LIN {X 0,Y 424.984,Z 508.898,A -85,B 0,C 180,E1 -17595.591,E2 -17595.591} C_VEL
LIN {X 0,Y 428.551,Z 453.272,A -85,B 0,C 180,E1 -17596.618,E2 -17596.618} C_VEL
LIN {X 0,Y 430.849,Z 412.705,A -85,B 0,C 180,E1 -17597.315,E2 -17597.315} C_VEL
LIN {X 0,Y 437.854,Z 381.493,A -85,B 0,C 180,E1 -17598.457,E2 -17598.457} C_VEL
LIN {X 0,Y 438.102,Z 374.288,A -85,B 0,C 180,E1 -17598.991,E2 -17598.991} C_VEL
LIN {X 0,Y 431.7,Z 356.101,A -85,B 0,C 180,E1 -17601.63,E2 -17601.63} C_VEL
LIN {X 0,Y 425.544,Z 340.551,A -85,B 0,C 180,E1 -17604.192,E2 -17604.192} C_VEL
LIN {X 0,Y 418.875,Z 325.42,A -85,B 0,C 180,E1 -17607.026,E2 -17607.026} C_VEL
LIN {X 0,Y 411.539,Z 310.81,A -85,B 0,C 180,E1 -17610.127,E2 -17610.127} C_VEL
LIN {X 0,Y 405.656,Z 300.356,A -85,B 0,C 180,E1 -17612.712,E2 -17612.712} C_VEL
LIN {X 0,Y 401.04,Z 292.309,A -85,B 0,C 180,E1 -17614.922,E2 -17614.922} C_VEL
LIN {X 0,Y 397.213,Z 286.474,A -85,B 0,C 180,E1 -17616.721,E2 -17616.721} C_VEL
LIN {X 0,Y 394.441,Z 281.986,A -85,B 0,C 180,E1 -17618.2,E2 -17618.2} C_VEL
LIN {X 0,Y 391.017,Z 276.874,A -85,B 0,C 180,E1 -17620.039,E2 -17620.039} C_VEL
LIN {X 0,Y 388.14,Z 272.719,A -85,B 0,C 180,E1 -17621.721,E2 -17621.721} C_VEL
LIN {X 0,Y 387.304,Z 271.349,A -85,B 0,C 180,E1 -17622.264,E2 -17622.264} C_VEL
LIN {X 0,Y 384.465,Z 267.744,A -85,B 0,C 180,E1 -17624.075,E2 -17624.075} C_VEL
LIN {X 0,Y 383.391,Z 265.721,A -85,B 0,C 180,E1 -17624.882,E2 -17624.882} C_VEL
LIN {X 0,Y 380.512,Z 262.705,A -85,B 0,C 180,E1 -17626.939,E2 -17626.939} C_VEL
LIN {X 0,Y 379.113,Z 259.666,A -85,B 0,C 180,E1 -17628.283,E2 -17628.283} C_VEL
LIN {X 0,Y 375.9,Z 257.035,A -85,B 0,C 180,E1 -17631.125,E2 -17631.125} C_VEL
LIN {X 0,Y 374.343,Z 253.325,A -85,B 0,C 180,E1 -17633.405,E2 -17633.405} C_VEL
LIN {X 0,Y 370.867,Z 250.89,A -85,B 0,C 180,E1 -17641.236,E2 -17641.236} C_VEL
LIN {X 0,Y 371.49,Z 251.549,A -85,B 0,C 180,E1 -17645.87,E2 -17645.87} C_VEL
LIN {X 0,Y 374.488,Z 253.671,A -85,B 0,C 180,E1 -17650.729,E2 -17650.729} C_VEL
LIN {X 0,Y 376.122,Z 261.606,A -85,B 0,C 180,E1 -17653.647,E2 -17653.647} C_VEL
LIN {X 0,Y 378.615,Z 269.925,A -85,B 0,C 180,E1 -17656.414,E2 -17656.414} C_VEL
LIN {X 0,Y 385.424,Z 282.96,A -85,B 0,C 180,E1 -17659.71,E2 -17659.71} C_VEL
LIN {X 0,Y 393.512,Z 298.865,A -85,B 0,C 180,E1 -17663.353,E2 -17663.353} C_VEL
LIN {X 0,Y 402.331,Z 316.84,A -85,B 0,C 180,E1 -17667.052,E2 -17667.052} C_VEL
LIN {X 0,Y 410.157,Z 332.928,A -85,B 0,C 180,E1 -17670.004,E2 -17670.004} C_VEL
LIN {X 0,Y 428.238,Z 360.802,A -85,B 0,C 180,E1 -17673.138,E2 -17673.138} C_VEL
LIN {X 0,Y 436.471,Z 374.047,A -85,B 0,C 180,E1 -17674.486,E2 -17674.486} C_VEL
LIN {X 0,Y 417.243,Z 631.491,A -85,B 0,C 180,E1 -17679.901,E2 -17679.901} C_VEL
LIN {X 0,Y 412.894,Z 693.948,A -85,B 0,C 180,E1 -17681.283,E2 -17681.283} C_VEL
LIN {X 0,Y 410.167,Z 718.357,A -85,B 0,C 180,E1 -17682.04,E2 -17682.04} C_VEL
LIN {X 0,Y 406.626,Z 743.879,A -85,B 0,C 180,E1 -17683.087,E2 -17683.087} C_VEL
LIN {X 0,Y 402.884,Z 766.939,A -85,B 0,C 180,E1 -17684.276,E2 -17684.276} C_VEL
LIN {X 0,Y 398.654,Z 789.481,A -85,B 0,C 180,E1 -17685.718,E2 -17685.718} C_VEL
LIN {X 0,Y 393.831,Z 812.889,A -85,B 0,C 180,E1 -17687.519,E2 -17687.519} C_VEL
LIN {X 0,Y 389.308,Z 833.205,A -85,B 0,C 180,E1 -17689.377,E2 -17689.377} C_VEL
LIN {X 0,Y 384.718,Z 852.523,A -85,B 0,C 180,E1 -17691.473,E2 -17691.473} C_VEL
LIN {X 0,Y 380.138,Z 871.424,A -85,B 0,C 180,E1 -17693.854,E2 -17693.854} C_VEL
LIN {X 0,Y 375.883,Z 888.627,A -85,B 0,C 180,E1 -17696.406,E2 -17696.406} C_VEL
LIN {X 0,Y 371.678,Z 905.948,A -85,B 0,C 180,E1 -17699.414,E2 -17699.414} C_VEL
LIN {X 0,Y 368.526,Z 919.642,A -85,B 0,C 180,E1 -17702.192,E2 -17702.192} C_VEL
LIN {X 0,Y 365.762,Z 932.567,A -85,B 0,C 180,E1 -17705.275,E2 -17705.275} C_VEL
LIN {X 0,Y 363.603,Z 944.291,A -85,B 0,C 180,E1 -17708.547,E2 -17708.547} C_VEL
LIN {X 0,Y 362.169,Z 953.987,A -85,B 0,C 180,E1 -17711.822,E2 -17711.822} C_VEL
LIN {X 0,Y 361.326,Z 962.067,A -85,B 0,C 180,E1 -17715.087,E2 -17715.087} C_VEL
LIN {X 0,Y 360.957,Z 968.703,A -85,B 0,C 180,E1 -17718.495,E2 -17718.495} C_VEL
LIN {X 0,Y 360.949,Z 973.188,A -85,B 0,C 180,E1 -17721.477,E2 -17721.477} C_VEL
LIN {X 0,Y 361.102,Z 976.867,A -85,B 0,C 180,E1 -17724.917,E2 -17724.917} C_VEL
LIN {X 0,Y 361.251,Z 978.684,A -85,B 0,C 180,E1 -17728.097,E2 -17728.097} C_VEL
LIN {X 0,Y 361.231,Z 979.16,A -85,B 0,C 180,E1 -17730.952,E2 -17730.952} C_VEL
LIN {X 0,Y 361.074,Z 978.468,A -85,B 0,C 180,E1 -17733.97,E2 -17733.97} C_VEL
LIN {X 0,Y 360.804,Z 976.089,A -85,B 0,C 180,E1 -17737.484,E2 -17737.484} C_VEL
LIN {X 0,Y 360.711,Z 972.725,A -85,B 0,C 180,E1 -17740.542,E2 -17740.542} C_VEL
LIN {X 0,Y 360.927,Z 967.69,A -85,B 0,C 180,E1 -17743.947,E2 -17743.947} C_VEL
LIN {X 0,Y 361.857,Z 960.075,A -85,B 0,C 180,E1 -17747.862,E2 -17747.862} C_VEL
LIN {X 0,Y 363.44,Z 951.875,A -85,B 0,C 180,E1 -17751.294,E2 -17751.294} C_VEL
LIN {X 0,Y 366.317,Z 940.57,A -85,B 0,C 180,E1 -17755.202,E2 -17755.202} C_VEL
LIN {X 0,Y 370.299,Z 927.832,A -85,B 0,C 180,E1 -17758.904,E2 -17758.904} C_VEL
LIN {X 0,Y 375.296,Z 913.565,A -85,B 0,C 180,E1 -17762.379,E2 -17762.379} C_VEL
LIN {X 0,Y 381.882,Z 896.522,A -85,B 0,C 180,E1 -17765.91,E2 -17765.91} C_VEL
LIN {X 0,Y 389.169,Z 878.862,A -85,B 0,C 180,E1 -17769.012,E2 -17769.012} C_VEL
LIN {X 0,Y 397.276,Z 859.703,A -85,B 0,C 180,E1 -17771.841,E2 -17771.841} C_VEL
LIN {X 0,Y 406.471,Z 838.288,A -85,B 0,C 180,E1 -17774.514,E2 -17774.514} C_VEL
LIN {X 0,Y 416.369,Z 815.377,A -85,B 0,C 180,E1 -17776.89,E2 -17776.89} C_VEL
LIN {X 0,Y 425.924,Z 793.069,A -85,B 0,C 180,E1 -17778.799,E2 -17778.799} C_VEL
LIN {X 0,Y 435.049,Z 771.007,A -85,B 0,C 180,E1 -17780.349,E2 -17780.349} C_VEL
LIN {X 0,Y 443.884,Z 748.687,A -85,B 0,C 180,E1 -17781.619,E2 -17781.619} C_VEL
LIN {X 0,Y 448.557,Z 736.3,A -85,B 0,C 180,E1 -17782.233,E2 -17782.233} C_VEL
LIN {X 0,Y 438.455,Z 757.223,A -85,B 0,C 180,E1 -17783.472,E2 -17783.472} C_VEL
LIN {X 0,Y 428.026,Z 777.505,A -85,B 0,C 180,E1 -17785.005,E2 -17785.005} C_VEL
LIN {X 0,Y 417.47,Z 797.566,A -85,B 0,C 180,E1 -17786.901,E2 -17786.901} C_VEL
LIN {X 0,Y 407.438,Z 816.792,A -85,B 0,C 180,E1 -17789.142,E2 -17789.142} C_VEL
LIN {X 0,Y 398.353,Z 834.637,A -85,B 0,C 180,E1 -17791.679,E2 -17791.679} C_VEL
LIN {X 0,Y 390.604,Z 850.206,A -85,B 0,C 180,E1 -17794.366,E2 -17794.366} C_VEL
LIN {X 0,Y 384.339,Z 862.875,A -85,B 0,C 180,E1 -17797.031,E2 -17797.031} C_VEL
LIN {X 0,Y 379.023,Z 873.475,A -85,B 0,C 180,E1 -17799.782,E2 -17799.782} C_VEL
LIN {X 0,Y 374.57,Z 882.04,A -85,B 0,C 180,E1 -17802.604,E2 -17802.604} C_VEL
LIN {X 0,Y 370.918,Z 888.625,A -85,B 0,C 180,E1 -17805.481,E2 -17805.481} C_VEL
LIN {X 0,Y 368.15,Z 893.065,A -85,B 0,C 180,E1 -17808.247,E2 -17808.247} C_VEL
LIN {X 0,Y 366.013,Z 895.825,A -85,B 0,C 180,E1 -17811.042,E2 -17811.042} C_VEL
LIN {X 0,Y 364.426,Z 896.884,A -85,B 0,C 180,E1 -17813.857,E2 -17813.857} C_VEL
LIN {X 0,Y 363.265,Z 896.126,A -85,B 0,C 180,E1 -17816.844,E2 -17816.844} C_VEL
LIN {X 0,Y 362.594,Z 893.619,A -85,B 0,C 180,E1 -17819.684,E2 -17819.684} C_VEL
LIN {X 0,Y 362.254,Z 889.408,A -85,B 0,C 180,E1 -17822.531,E2 -17822.531} C_VEL
LIN {X 0,Y 362.232,Z 883.769,A -85,B 0,C 180,E1 -17825.226,E2 -17825.226} C_VEL
LIN {X 0,Y 362.532,Z 875.956,A -85,B 0,C 180,E1 -17828.086,E2 -17828.086} C_VEL
LIN {X 0,Y 363.206,Z 866.063,A -85,B 0,C 180,E1 -17830.95,E2 -17830.95} C_VEL
LIN {X 0,Y 364.27,Z 854.546,A -85,B 0,C 180,E1 -17833.663,E2 -17833.663} C_VEL
LIN {X 0,Y 365.672,Z 841.577,A -85,B 0,C 180,E1 -17836.195,E2 -17836.195} C_VEL
LIN {X 0,Y 367.459,Z 826.606,A -85,B 0,C 180,E1 -17838.647,E2 -17838.647} C_VEL
LIN {X 0,Y 369.541,Z 810.047,A -85,B 0,C 180,E1 -17840.926,E2 -17840.926} C_VEL
LIN {X 0,Y 371.846,Z 791.943,A -85,B 0,C 180,E1 -17843.012,E2 -17843.012} C_VEL
LIN {X 0,Y 374.252,Z 772.49,A -85,B 0,C 180,E1 -17844.885,E2 -17844.885} C_VEL
LIN {X 0,Y 376.791,Z 751.357,A -85,B 0,C 180,E1 -17846.561,E2 -17846.561} C_VEL
LIN {X 0,Y 379.246,Z 729.129,A -85,B 0,C 180,E1 -17847.989,E2 -17847.989} C_VEL
LIN {X 0,Y 381.469,Z 706.375,A -85,B 0,C 180,E1 -17849.137,E2 -17849.137} C_VEL
LIN {X 0,Y 383.428,Z 682.672,A -85,B 0,C 180,E1 -17850.019,E2 -17850.019} C_VEL
LIN {X 0,Y 395.248,Z 511.536,A -85,B 0,C 180,E1 -17854.648,E2 -17854.648} C_VEL
LIN {X 0,Y 391.838,Z 447.433,A -85,B 0,C 180,E1 -17857.121,E2 -17857.121} C_VEL
LIN {X 0,Y 393.218,Z 446.968,A -85,B 0,C 180,E1 -17857.381,E2 -17857.381} C_VEL
LIN {X 0,Y 395.398,Z 443.797,A -85,B 0,C 180,E1 -17857.71,E2 -17857.71} C_VEL
LIN {X 0,Y 398.815,Z 435.862,A -85,B 0,C 180,E1 -17858.126,E2 -17858.126} C_VEL
LIN {X 0,Y 400.426,Z 433.355,A -85,B 0,C 180,E1 -17858.354,E2 -17858.354} C_VEL
LIN {X 0,Y 404.177,Z 431.028,A -85,B 0,C 180,E1 -17858.976,E2 -17858.976} C_VEL
LIN {X 0,Y 408.609,Z 426.161,A -85,B 0,C 180,E1 -17859.626,E2 -17859.626} C_VEL
LIN {X 0,Y 409.577,Z 425.061,A -85,B 0,C 180,E1 -17859.763,E2 -17859.763} C_VEL
LIN {X 0,Y 414.152,Z 421.888,A -85,B 0,C 180,E1 -17860.455,E2 -17860.455} C_VEL
LIN {X 0,Y 418.92,Z 417.332,A -85,B 0,C 180,E1 -17861.025,E2 -17861.025} C_VEL
LIN {X 0,Y 423.934,Z 414.013,A -85,B 0,C 180,E1 -17861.692,E2 -17861.692} C_VEL
LIN {X 0,Y 428.557,Z 410.023,A -85,B 0,C 180,E1 -17862.218,E2 -17862.218} C_VEL
LIN {X 0,Y 431.714,Z 408.162,A -85,B 0,C 180,E1 -17862.628,E2 -17862.628} C_VEL
LIN {X 0,Y 430.489,Z 414.914,A -85,B 0,C 180,E1 -17862.841,E2 -17862.841} C_VEL
LIN {X 0,Y 425.936,Z 494.183,A -85,B 0,C 180,E1 -17864.222,E2 -17864.222} C_VEL
LIN {X 0,Y 421.205,Z 553.034,A -85,B 0,C 180,E1 -17865.466,E2 -17865.466} C_VEL
LIN {X 0,Y 415.261,Z 612.433,A -85,B 0,C 180,E1 -17866.95,E2 -17866.95} C_VEL
LIN {X 0,Y 410.707,Z 656.621,A -85,B 0,C 180,E1 -17868.27,E2 -17868.27} C_VEL
LIN {X 0,Y 408.041,Z 685.292,A -85,B 0,C 180,E1 -17869.326,E2 -17869.326} C_VEL
LIN {X 0,Y 405.524,Z 705.596,A -85,B 0,C 180,E1 -17870.312,E2 -17870.312} C_VEL
LIN {X 0,Y 402.242,Z 726.337,A -85,B 0,C 180,E1 -17871.578,E2 -17871.578} C_VEL
LIN {X 0,Y 398.508,Z 746.053,A -85,B 0,C 180,E1 -17873.064,E2 -17873.064} C_VEL
LIN {X 0,Y 394.229,Z 765.506,A -85,B 0,C 180,E1 -17874.848,E2 -17874.848} C_VEL
LIN {X 0,Y 389.705,Z 783.802,A -85,B 0,C 180,E1 -17876.872,E2 -17876.872} C_VEL
LIN {X 0,Y 385.137,Z 800.764,A -85,B 0,C 180,E1 -17879.122,E2 -17879.122} C_VEL
LIN {X 0,Y 380.552,Z 816.747,A -85,B 0,C 180,E1 -17881.668,E2 -17881.668} C_VEL
LIN {X 0,Y 376.385,Z 830.752,A -85,B 0,C 180,E1 -17884.341,E2 -17884.341} C_VEL
LIN {X 0,Y 372.544,Z 843.468,A -85,B 0,C 180,E1 -17887.264,E2 -17887.264} C_VEL
LIN {X 0,Y 369.226,Z 854.588,A -85,B 0,C 180,E1 -17890.379,E2 -17890.379} C_VEL
LIN {X 0,Y 366.629,Z 863.669,A -85,B 0,C 180,E1 -17893.523,E2 -17893.523} C_VEL
LIN {X 0,Y 364.673,Z 871.061,A -85,B 0,C 180,E1 -17896.749,E2 -17896.749} C_VEL
LIN {X 0,Y 363.308,Z 876.769,A -85,B 0,C 180,E1 -17900.015,E2 -17900.015} C_VEL
LIN {X 0,Y 362.432,Z 881.033,A -85,B 0,C 180,E1 -17903.505,E2 -17903.505} C_VEL
LIN {X 0,Y 362.034,Z 883.325,A -85,B 0,C 180,E1 -17906.583,E2 -17906.583} C_VEL
LIN {X 0,Y 360.957,Z 883.954,A -85,B 0,C 180,E1 -17907.799,E2 -17907.799} C_VEL
LIN {X 0,Y 354.617,Z 885.109,A -85,B 0,C 180,E1 -17911.143,E2 -17911.143} C_VEL
LIN {X 0,Y 354.012,Z 884.908,A -85,B 0,C 180,E1 -17912.13,E2 -17912.13} C_VEL
LIN {X 0,Y 354.34,Z 883.134,A -85,B 0,C 180,E1 -17915.505,E2 -17915.505} C_VEL
LIN {X 0,Y 355.032,Z 879.694,A -85,B 0,C 180,E1 -17918.911,E2 -17918.911} C_VEL
LIN {X 0,Y 356.194,Z 874.854,A -85,B 0,C 180,E1 -17922.154,E2 -17922.154} C_VEL
LIN {X 0,Y 358.029,Z 868.036,A -85,B 0,C 180,E1 -17925.551,E2 -17925.551} C_VEL
LIN {X 0,Y 360.466,Z 859.76,A -85,B 0,C 180,E1 -17928.77,E2 -17928.77} C_VEL
LIN {X 0,Y 363.449,Z 850.138,A -85,B 0,C 180,E1 -17931.802,E2 -17931.802} C_VEL
LIN {X 0,Y 367.117,Z 838.547,A -85,B 0,C 180,E1 -17934.799,E2 -17934.799} C_VEL
LIN {X 0,Y 371.487,Z 824.659,A -85,B 0,C 180,E1 -17937.752,E2 -17937.752} C_VEL
LIN {X 0,Y 376.128,Z 809.477,A -85,B 0,C 180,E1 -17940.426,E2 -17940.426} C_VEL
LIN {X 0,Y 380.722,Z 793.669,A -85,B 0,C 180,E1 -17942.753,E2 -17942.753} C_VEL
LIN {X 0,Y 385.565,Z 775.624,A -85,B 0,C 180,E1 -17944.968,E2 -17944.968} C_VEL
LIN {X 0,Y 390.072,Z 757.084,A -85,B 0,C 180,E1 -17946.857,E2 -17946.857} C_VEL
LIN {X 0,Y 394.24,Z 737.467,A -85,B 0,C 180,E1 -17948.51,E2 -17948.51} C_VEL
LIN {X 0,Y 397.983,Z 716.674,A -85,B 0,C 180,E1 -17949.935,E2 -17949.935} C_VEL
LIN {X 0,Y 401.085,Z 695.03,A -85,B 0,C 180,E1 -17951.117,E2 -17951.117} C_VEL
LIN {X 0,Y 403.458,Z 672.77,A -85,B 0,C 180,E1 -17952.049,E2 -17952.049} C_VEL
LIN {X 0,Y 407.778,Z 629.715,A -85,B 0,C 180,E1 -17953.455,E2 -17953.455} C_VEL
LIN {X 0,Y 414.06,Z 571.27,A -85,B 0,C 180,E1 -17955.005,E2 -17955.005} C_VEL
LIN {X 0,Y 419.279,Z 512.395,A -85,B 0,C 180,E1 -17956.318,E2 -17956.318} C_VEL
LIN {X 0,Y 422.898,Z 458.138,A -85,B 0,C 180,E1 -17957.334,E2 -17957.334} C_VEL
LIN {X 0,Y 425.379,Z 415.515,A -85,B 0,C 180,E1 -17958.07,E2 -17958.07} C_VEL
LIN {X 0,Y 432.668,Z 383.274,A -85,B 0,C 180,E1 -17959.238,E2 -17959.238} C_VEL
LIN {X 0,Y 432.805,Z 378.392,A -85,B 0,C 180,E1 -17959.607,E2 -17959.607} C_VEL
LIN {X 0,Y 426.533,Z 360.369,A -85,B 0,C 180,E1 -17962.277,E2 -17962.277} C_VEL
LIN {X 0,Y 420.306,Z 344.672,A -85,B 0,C 180,E1 -17964.921,E2 -17964.921} C_VEL
LIN {X 0,Y 413.62,Z 329.35,A -85,B 0,C 180,E1 -17967.871,E2 -17967.871} C_VEL
LIN {X 0,Y 407.095,Z 316.323,A -85,B 0,C 180,E1 -17970.74,E2 -17970.74} C_VEL
LIN {X 0,Y 401.641,Z 306.431,A -85,B 0,C 180,E1 -17973.217,E2 -17973.217} C_VEL
LIN {X 0,Y 397.019,Z 298.327,A -85,B 0,C 180,E1 -17975.525,E2 -17975.525} C_VEL
LIN {X 0,Y 393.875,Z 293.356,A -85,B 0,C 180,E1 -17977.066,E2 -17977.066} C_VEL
LIN {X 0,Y 391.222,Z 288.934,A -85,B 0,C 180,E1 -17978.563,E2 -17978.563} C_VEL
LIN {X 0,Y 387.999,Z 284.027,A -85,B 0,C 180,E1 -17980.348,E2 -17980.348} C_VEL
LIN {X 0,Y 385.133,Z 279.626,A -85,B 0,C 180,E1 -17982.121,E2 -17982.121} C_VEL
LIN {X 0,Y 381.484,Z 274.487,A -85,B 0,C 180,E1 -17984.571,E2 -17984.571} C_VEL
LIN {X 0,Y 380.825,Z 273.211,A -85,B 0,C 180,E1 -17985.09,E2 -17985.09} C_VEL
LIN {X 0,Y 377.944,Z 270.024,A -85,B 0,C 180,E1 -17987.238,E2 -17987.238} C_VEL
LIN {X 0,Y 376.766,Z 267.259,A -85,B 0,C 180,E1 -17988.519,E2 -17988.519} C_VEL
LIN {X 0,Y 373.477,Z 264.326,A -85,B 0,C 180,E1 -17991.532,E2 -17991.532} C_VEL
LIN {X 0,Y 372.123,Z 260.992,A -85,B 0,C 180,E1 -17993.675,E2 -17993.675} C_VEL
LIN {X 0,Y 369.027,Z 258.675,A -85,B 0,C 180,E1 -18001.242,E2 -18001.242} C_VEL
LIN {X 0,Y 369.744,Z 259.37,A -85,B 0,C 180,E1 -18005.898,E2 -18005.898} C_VEL
LIN {X 0,Y 372.489,Z 261.356,A -85,B 0,C 180,E1 -18010.439,E2 -18010.439} C_VEL
LIN {X 0,Y 373.965,Z 268.68,A -85,B 0,C 180,E1 -18013.176,E2 -18013.176} C_VEL
LIN {X 0,Y 376.51,Z 277.821,A -85,B 0,C 180,E1 -18016.191,E2 -18016.191} C_VEL
LIN {X 0,Y 381.85,Z 292.334,A -85,B 0,C 180,E1 -18020.381,E2 -18020.381} C_VEL
LIN {X 0,Y 390.043,Z 308.671,A -85,B 0,C 180,E1 -18024.054,E2 -18024.054} C_VEL
LIN {X 0,Y 399.158,Z 327.437,A -85,B 0,C 180,E1 -18027.839,E2 -18027.839} C_VEL
LIN {X 0,Y 402.379,Z 333.924,A -85,B 0,C 180,E1 -18029.01,E2 -18029.01} C_VEL
LIN {X 0,Y 422.571,Z 365.09,A -85,B 0,C 180,E1 -18032.601,E2 -18032.601} C_VEL
LIN {X 0,Y 430.139,Z 377.336,A -85,B 0,C 180,E1 -18033.862,E2 -18033.862} C_VEL
LIN {X 0,Y 410.702,Z 628.411,A -85,B 0,C 180,E1 -18039.24,E2 -18039.24} C_VEL
LIN {X 0,Y 405.985,Z 693.922,A -85,B 0,C 180,E1 -18040.718,E2 -18040.718} C_VEL
LIN {X 0,Y 403.21,Z 718.115,A -85,B 0,C 180,E1 -18041.482,E2 -18041.482} C_VEL
LIN {X 0,Y 399.697,Z 742.919,A -85,B 0,C 180,E1 -18042.511,E2 -18042.511} C_VEL
LIN {X 0,Y 395.798,Z 766.429,A -85,B 0,C 180,E1 -18043.738,E2 -18043.738} C_VEL
LIN {X 0,Y 391.526,Z 788.691,A -85,B 0,C 180,E1 -18045.182,E2 -18045.182} C_VEL
LIN {X 0,Y 386.728,Z 811.509,A -85,B 0,C 180,E1 -18046.955,E2 -18046.955} C_VEL
LIN {X 0,Y 382.094,Z 831.899,A -85,B 0,C 180,E1 -18048.842,E2 -18048.842} C_VEL
LIN {X 0,Y 377.316,Z 851.634,A -85,B 0,C 180,E1 -18051.002,E2 -18051.002} C_VEL
LIN {X 0,Y 372.803,Z 869.858,A -85,B 0,C 180,E1 -18053.317,E2 -18053.317} C_VEL
LIN {X 0,Y 368.526,Z 886.743,A -85,B 0,C 180,E1 -18055.846,E2 -18055.846} C_VEL
LIN {X 0,Y 364.361,Z 903.466,A -85,B 0,C 180,E1 -18058.758,E2 -18058.758} C_VEL
LIN {X 0,Y 361.088,Z 917.18,A -85,B 0,C 180,E1 -18061.557,E2 -18061.557} C_VEL
LIN {X 0,Y 358.024,Z 931.1,A -85,B 0,C 180,E1 -18064.881,E2 -18064.881} C_VEL
LIN {X 0,Y 355.871,Z 942.358,A -85,B 0,C 180,E1 -18068.057,E2 -18068.057} C_VEL
LIN {X 0,Y 354.277,Z 952.735,A -85,B 0,C 180,E1 -18071.573,E2 -18071.573} C_VEL
LIN {X 0,Y 353.4,Z 960.861,A -85,B 0,C 180,E1 -18074.912,E2 -18074.912} C_VEL
LIN {X 0,Y 353.012,Z 967.793,A -85,B 0,C 180,E1 -18078.531,E2 -18078.531} C_VEL
LIN {X 0,Y 353.017,Z 972.197,A -85,B 0,C 180,E1 -18081.53,E2 -18081.53} C_VEL
LIN {X 0,Y 353.177,Z 975.815,A -85,B 0,C 180,E1 -18084.965,E2 -18084.965} C_VEL
LIN {X 0,Y 353.328,Z 977.637,A -85,B 0,C 180,E1 -18088.216,E2 -18088.216} C_VEL
LIN {X 0,Y 353.299,Z 978.106,A -85,B 0,C 180,E1 -18091.135,E2 -18091.135} C_VEL
LIN {X 0,Y 353.106,Z 977.399,A -85,B 0,C 180,E1 -18094.222,E2 -18094.222} C_VEL
LIN {X 0,Y 352.83,Z 975.02,A -85,B 0,C 180,E1 -18097.818,E2 -18097.818} C_VEL
LIN {X 0,Y 352.727,Z 971.431,A -85,B 0,C 180,E1 -18101.114,E2 -18101.114} C_VEL
LIN {X 0,Y 353.03,Z 966.335,A -85,B 0,C 180,E1 -18104.601,E2 -18104.601} C_VEL
LIN {X 0,Y 354.059,Z 959.013,A -85,B 0,C 180,E1 -18108.439,E2 -18108.439} C_VEL
LIN {X 0,Y 355.906,Z 950.42,A -85,B 0,C 180,E1 -18112.115,E2 -18112.115} C_VEL
LIN {X 0,Y 359.099,Z 939.101,A -85,B 0,C 180,E1 -18116.1,E2 -18116.1} C_VEL
LIN {X 0,Y 363.454,Z 926.402,A -85,B 0,C 180,E1 -18119.864,E2 -18119.864} C_VEL
LIN {X 0,Y 368.927,Z 912.1,A -85,B 0,C 180,E1 -18123.408,E2 -18123.408} C_VEL
LIN {X 0,Y 375.947,Z 895.333,A -85,B 0,C 180,E1 -18126.948,E2 -18126.948} C_VEL
LIN {X 0,Y 383.727,Z 877.917,A -85,B 0,C 180,E1 -18130.062,E2 -18130.062} C_VEL
LIN {X 0,Y 392.756,Z 858.185,A -85,B 0,C 180,E1 -18133.023,E2 -18133.023} C_VEL
LIN {X 0,Y 402.833,Z 836.606,A -85,B 0,C 180,E1 -18135.734,E2 -18135.734} C_VEL
LIN {X 0,Y 413.334,Z 814.204,A -85,B 0,C 180,E1 -18138.062,E2 -18138.062} C_VEL
LIN {X 0,Y 423.737,Z 791.887,A -85,B 0,C 180,E1 -18139.971,E2 -18139.971} C_VEL
LIN {X 0,Y 433.523,Z 770.179,A -85,B 0,C 180,E1 -18141.484,E2 -18141.484} C_VEL
LIN {X 0,Y 439.331,Z 756.867,A -85,B 0,C 180,E1 -18142.29,E2 -18142.29} C_VEL
LIN {X 0,Y 428.322,Z 776.559,A -85,B 0,C 180,E1 -18143.716,E2 -18143.716} C_VEL
LIN {X 0,Y 416.856,Z 796.27,A -85,B 0,C 180,E1 -18145.522,E2 -18145.522} C_VEL
LIN {X 0,Y 405.872,Z 815.235,A -85,B 0,C 180,E1 -18147.684,E2 -18147.684} C_VEL
LIN {X 0,Y 395.858,Z 832.952,A -85,B 0,C 180,E1 -18150.159,E2 -18150.159} C_VEL
LIN {X 0,Y 387.233,Z 848.533,A -85,B 0,C 180,E1 -18152.804,E2 -18152.804} C_VEL
LIN {X 0,Y 379.645,Z 862.38,A -85,B 0,C 180,E1 -18155.683,E2 -18155.683} C_VEL
LIN {X 0,Y 373.638,Z 873.294,A -85,B 0,C 180,E1 -18158.492,E2 -18158.492} C_VEL
LIN {X 0,Y 368.676,Z 882.065,A -85,B 0,C 180,E1 -18161.335,E2 -18161.335} C_VEL
LIN {X 0,Y 364.771,Z 888.63,A -85,B 0,C 180,E1 -18164.091,E2 -18164.091} C_VEL
LIN {X 0,Y 361.266,Z 893.892,A -85,B 0,C 180,E1 -18167.208,E2 -18167.208} C_VEL
LIN {X 0,Y 358.703,Z 896.947,A -85,B 0,C 180,E1 -18170.21,E2 -18170.21} C_VEL
LIN {X 0,Y 356.898,Z 898.104,A -85,B 0,C 180,E1 -18173.081,E2 -18173.081} C_VEL
LIN {X 0,Y 355.611,Z 897.569,A -85,B 0,C 180,E1 -18175.969,E2 -18175.969} C_VEL
LIN {X 0,Y 354.79,Z 895.361,A -85,B 0,C 180,E1 -18178.87,E2 -18178.87} C_VEL
LIN {X 0,Y 354.351,Z 891.466,A -85,B 0,C 180,E1 -18181.779,E2 -18181.779} C_VEL
LIN {X 0,Y 354.245,Z 885.77,A -85,B 0,C 180,E1 -18184.695,E2 -18184.695} C_VEL
LIN {X 0,Y 354.468,Z 878.694,A -85,B 0,C 180,E1 -18187.456,E2 -18187.456} C_VEL
LIN {X 0,Y 355.018,Z 869.756,A -85,B 0,C 180,E1 -18190.221,E2 -18190.221} C_VEL
LIN {X 0,Y 355.971,Z 858.79,A -85,B 0,C 180,E1 -18192.986,E2 -18192.986} C_VEL
LIN {X 0,Y 357.29,Z 846.403,A -85,B 0,C 180,E1 -18195.585,E2 -18195.585} C_VEL
LIN {X 0,Y 358.979,Z 832.235,A -85,B 0,C 180,E1 -18198.081,E2 -18198.081} C_VEL
LIN {X 0,Y 360.984,Z 816.384,A -85,B 0,C 180,E1 -18200.427,E2 -18200.427} C_VEL
LIN {X 0,Y 363.327,Z 798.388,A -85,B 0,C 180,E1 -18202.662,E2 -18202.662} C_VEL
LIN {X 0,Y 365.876,Z 778.547,A -85,B 0,C 180,E1 -18204.717,E2 -18204.717} C_VEL
LIN {X 0,Y 368.373,Z 758.536,A -85,B 0,C 180,E1 -18206.433,E2 -18206.433} C_VEL
LIN {X 0,Y 370.948,Z 736.616,A -85,B 0,C 180,E1 -18207.971,E2 -18207.971} C_VEL
LIN {X 0,Y 373.29,Z 714.104,A -85,B 0,C 180,E1 -18209.221,E2 -18209.221} C_VEL
LIN {X 0,Y 375.438,Z 690.485,A -85,B 0,C 180,E1 -18210.222,E2 -18210.222} C_VEL
LIN {X 0,Y 378.003,Z 654.561,A -85,B 0,C 180,E1 -18211.312,E2 -18211.312} C_VEL
LIN {X 0,Y 388.249,Z 512.214,A -85,B 0,C 180,E1 -18215.216,E2 -18215.216} C_VEL
LIN {X 0,Y 386.223,Z 472.757,A -85,B 0,C 180,E1 -18216.776,E2 -18216.776} C_VEL
LIN {X 0,Y 387.587,Z 472.354,A -85,B 0,C 180,E1 -18217.041,E2 -18217.041} C_VEL
LIN {X 0,Y 389.842,Z 469.038,A -85,B 0,C 180,E1 -18217.39,E2 -18217.39} C_VEL
LIN {X 0,Y 392.918,Z 461.347,A -85,B 0,C 180,E1 -18217.759,E2 -18217.759} C_VEL
LIN {X 0,Y 395.267,Z 453.532,A -85,B 0,C 180,E1 -18217.977,E2 -18217.977} C_VEL
LIN {X 0,Y 398.142,Z 449.735,A -85,B 0,C 180,E1 -18218.409,E2 -18218.409} C_VEL
LIN {X 0,Y 401.43,Z 442.671,A -85,B 0,C 180,E1 -18218.811,E2 -18218.811} C_VEL
LIN {X 0,Y 402.505,Z 440.316,A -85,B 0,C 180,E1 -18218.939,E2 -18218.939} C_VEL
LIN {X 0,Y 407.194,Z 436.824,A -85,B 0,C 180,E1 -18219.676,E2 -18219.676} C_VEL
LIN {X 0,Y 411.77,Z 431.891,A -85,B 0,C 180,E1 -18220.326,E2 -18220.326} C_VEL
LIN {X 0,Y 417.125,Z 427.794,A -85,B 0,C 180,E1 -18221.103,E2 -18221.103} C_VEL
LIN {X 0,Y 421.231,Z 423.838,A -85,B 0,C 180,E1 -18221.655,E2 -18221.655} C_VEL
LIN {X 0,Y 424.807,Z 421.477,A -85,B 0,C 180,E1 -18222.151,E2 -18222.151} C_VEL
LIN {X 0,Y 420.272,Z 497.691,A -85,B 0,C 180,E1 -18223.49,E2 -18223.49} C_VEL
LIN {X 0,Y 415.453,Z 555.616,A -85,B 0,C 180,E1 -18224.729,E2 -18224.729} C_VEL
LIN {X 0,Y 409.469,Z 613.57,A -85,B 0,C 180,E1 -18226.194,E2 -18226.194} C_VEL
LIN {X 0,Y 404.775,Z 657.664,A -85,B 0,C 180,E1 -18227.528,E2 -18227.528} C_VEL
LIN {X 0,Y 401.93,Z 687.022,A -85,B 0,C 180,E1 -18228.627,E2 -18228.627} C_VEL
LIN {X 0,Y 399.248,Z 707.767,A -85,B 0,C 180,E1 -18229.654,E2 -18229.654} C_VEL
LIN {X 0,Y 395.858,Z 728.321,A -85,B 0,C 180,E1 -18230.934,E2 -18230.934} C_VEL
LIN {X 0,Y 392.003,Z 747.896,A -85,B 0,C 180,E1 -18232.438,E2 -18232.438} C_VEL
LIN {X 0,Y 387.583,Z 767.232,A -85,B 0,C 180,E1 -18234.244,E2 -18234.244} C_VEL
LIN {X 0,Y 382.853,Z 785.607,A -85,B 0,C 180,E1 -18236.318,E2 -18236.318} C_VEL
LIN {X 0,Y 378.121,Z 802.479,A -85,B 0,C 180,E1 -18238.604,E2 -18238.604} C_VEL
LIN {X 0,Y 373.387,Z 818.314,A -85,B 0,C 180,E1 -18241.182,E2 -18241.182} C_VEL
LIN {X 0,Y 368.975,Z 832.505,A -85,B 0,C 180,E1 -18243.959,E2 -18243.959} C_VEL
LIN {X 0,Y 364.997,Z 845.109,A -85,B 0,C 180,E1 -18246.937,E2 -18246.937} C_VEL
LIN {X 0,Y 361.557,Z 856.127,A -85,B 0,C 180,E1 -18250.113,E2 -18250.113} C_VEL
LIN {X 0,Y 358.734,Z 865.576,A -85,B 0,C 180,E1 -18253.501,E2 -18253.501} C_VEL
LIN {X 0,Y 356.696,Z 872.928,A -85,B 0,C 180,E1 -18256.876,E2 -18256.876} C_VEL
LIN {X 0,Y 355.302,Z 878.489,A -85,B 0,C 180,E1 -18260.279,E2 -18260.279} C_VEL
LIN {X 0,Y 354.473,Z 882.337,A -85,B 0,C 180,E1 -18263.684,E2 -18263.684} C_VEL
LIN {X 0,Y 354.056,Z 884.554,A -85,B 0,C 180,E1 -18267.086,E2 -18267.086} C_VEL
LIN {X 0,Y 353.956,Z 885.197,A -85,B 0,C 180,E1 -18270.324,E2 -18270.324} C_VEL
LIN {X 0,Y 354.012,Z 884.908,A -85,B 0,C 180,E1 -18272.13,E2 -18272.13} C_VEL
LIN {X 0,Y 353.105,Z 884.552,A -85,B 0,C 180,E1 -18273.378,E2 -18273.378} C_VEL
LIN {X 0,Y 347.381,Z 883.219,A -85,B 0,C 180,E1 -18276.728,E2 -18276.728} C_VEL
LIN {X 0,Y 346.846,Z 882.204,A -85,B 0,C 180,E1 -18277.815,E2 -18277.815} C_VEL
LIN {X 0,Y 347.975,Z 877.54,A -85,B 0,C 180,E1 -18281.436,E2 -18281.436} C_VEL
LIN {X 0,Y 349.824,Z 870.903,A -85,B 0,C 180,E1 -18285.076,E2 -18285.076} C_VEL
LIN {X 0,Y 352.418,Z 862.388,A -85,B 0,C 180,E1 -18288.623,E2 -18288.623} C_VEL
LIN {X 0,Y 355.68,Z 852.278,A -85,B 0,C 180,E1 -18291.956,E2 -18291.956} C_VEL
LIN {X 0,Y 359.439,Z 840.872,A -85,B 0,C 180,E1 -18295.014,E2 -18295.014} C_VEL
LIN {X 0,Y 363.671,Z 828.008,A -85,B 0,C 180,E1 -18297.866,E2 -18297.866} C_VEL
LIN {X 0,Y 367.962,Z 814.594,A -85,B 0,C 180,E1 -18300.36,E2 -18300.36} C_VEL
LIN {X 0,Y 372.603,Z 799.462,A -85,B 0,C 180,E1 -18302.733,E2 -18302.733} C_VEL
LIN {X 0,Y 377.344,Z 782.911,A -85,B 0,C 180,E1 -18304.915,E2 -18304.915} C_VEL
LIN {X 0,Y 381.724,Z 766.258,A -85,B 0,C 180,E1 -18306.765,E2 -18306.765} C_VEL
LIN {X 0,Y 385.962,Z 748.26,A -85,B 0,C 180,E1 -18308.444,E2 -18308.444} C_VEL
LIN {X 0,Y 389.967,Z 728.551,A -85,B 0,C 180,E1 -18309.963,E2 -18309.963} C_VEL
LIN {X 0,Y 393.455,Z 707.895,A -85,B 0,C 180,E1 -18311.25,E2 -18311.25} C_VEL
LIN {X 0,Y 396.308,Z 686.094,A -85,B 0,C 180,E1 -18312.318,E2 -18312.318} C_VEL
LIN {X 0,Y 399.857,Z 650.548,A -85,B 0,C 180,E1 -18313.613,E2 -18313.613} C_VEL
LIN {X 0,Y 405.349,Z 601.675,A -85,B 0,C 180,E1 -18315.044,E2 -18315.044} C_VEL
LIN {X 0,Y 410.919,Z 547.326,A -85,B 0,C 180,E1 -18316.384,E2 -18316.384} C_VEL
LIN {X 0,Y 415.551,Z 490.609,A -85,B 0,C 180,E1 -18317.569,E2 -18317.569} C_VEL
LIN {X 0,Y 419.979,Z 418.206,A -85,B 0,C 180,E1 -18318.845,E2 -18318.845} C_VEL
LIN {X 0,Y 427.547,Z 384.988,A -85,B 0,C 180,E1 -18320.04,E2 -18320.04} C_VEL
LIN {X 0,Y 427.552,Z 382.519,A -85,B 0,C 180,E1 -18320.236,E2 -18320.236} C_VEL
LIN {X 0,Y 421.414,Z 364.665,A -85,B 0,C 180,E1 -18322.939,E2 -18322.939} C_VEL
LIN {X 0,Y 415.15,Z 348.657,A -85,B 0,C 180,E1 -18325.702,E2 -18325.702} C_VEL
LIN {X 0,Y 408.377,Z 333.351,A -85,B 0,C 180,E1 -18328.73,E2 -18328.73} C_VEL
LIN {X 0,Y 402.415,Z 321.186,A -85,B 0,C 180,E1 -18331.506,E2 -18331.506} C_VEL
LIN {X 0,Y 396.611,Z 310.397,A -85,B 0,C 180,E1 -18334.302,E2 -18334.302} C_VEL
LIN {X 0,Y 391.135,Z 301.045,A -85,B 0,C 180,E1 -18337.134,E2 -18337.134} C_VEL
LIN {X 0,Y 388.021,Z 295.874,A -85,B 0,C 180,E1 -18338.932,E2 -18338.932} C_VEL
LIN {X 0,Y 384.994,Z 291.173,A -85,B 0,C 180,E1 -18340.662,E2 -18340.662} C_VEL
LIN {X 0,Y 382.188,Z 286.545,A -85,B 0,C 180,E1 -18342.53,E2 -18342.53} C_VEL
LIN {X 0,Y 378.955,Z 282.176,A -85,B 0,C 180,E1 -18344.701,E2 -18344.701} C_VEL
LIN {X 0,Y 378.03,Z 280.526,A -85,B 0,C 180,E1 -18345.447,E2 -18345.447} C_VEL
LIN {X 0,Y 375.234,Z 277.05,A -85,B 0,C 180,E1 -18347.691,E2 -18347.691} C_VEL
LIN {X 0,Y 374.296,Z 274.809,A -85,B 0,C 180,E1 -18348.755,E2 -18348.755} C_VEL
LIN {X 0,Y 371.321,Z 271.937,A -85,B 0,C 180,E1 -18351.717,E2 -18351.717} C_VEL
LIN {X 0,Y 370.039,Z 268.706,A -85,B 0,C 180,E1 -18353.795,E2 -18353.795} C_VEL
LIN {X 0,Y 367.154,Z 266.442,A -85,B 0,C 180,E1 -18361.404,E2 -18361.404} C_VEL
LIN {X 0,Y 368.011,Z 267.237,A -85,B 0,C 180,E1 -18366.083,E2 -18366.083} C_VEL
LIN {X 0,Y 370.532,Z 269.088,A -85,B 0,C 180,E1 -18370.181,E2 -18370.181} C_VEL
LIN {X 0,Y 371.851,Z 275.876,A -85,B 0,C 180,E1 -18372.738,E2 -18372.738} C_VEL
LIN {X 0,Y 374.308,Z 285.032,A -85,B 0,C 180,E1 -18375.772,E2 -18375.772} C_VEL
LIN {X 0,Y 379.498,Z 300.184,A -85,B 0,C 180,E1 -18380.151,E2 -18380.151} C_VEL
LIN {X 0,Y 387.563,Z 319.875,A -85,B 0,C 180,E1 -18384.868,E2 -18384.868} C_VEL
LIN {X 0,Y 394.603,Z 335.094,A -85,B 0,C 180,E1 -18387.996,E2 -18387.996} C_VEL
LIN {X 0,Y 411.937,Z 361.642,A -85,B 0,C 180,E1 -18391.193,E2 -18391.193} C_VEL
LIN {X 0,Y 423.773,Z 380.727,A -85,B 0,C 180,E1 -18393.234,E2 -18393.234} C_VEL
LIN {X 0,Y 403.08,Z 640.594,A -85,B 0,C 180,E1 -18398.906,E2 -18398.906} C_VEL
LIN {X 0,Y 398.994,Z 694.506,A -85,B 0,C 180,E1 -18400.166,E2 -18400.166} C_VEL
LIN {X 0,Y 396.142,Z 718.636,A -85,B 0,C 180,E1 -18400.946,E2 -18400.946} C_VEL
LIN {X 0,Y 392.53,Z 743.375,A -85,B 0,C 180,E1 -18401.998,E2 -18401.998} C_VEL
LIN {X 0,Y 388.52,Z 766.895,A -85,B 0,C 180,E1 -18403.254,E2 -18403.254} C_VEL
LIN {X 0,Y 383.956,Z 790.092,A -85,B 0,C 180,E1 -18404.795,E2 -18404.795} C_VEL
LIN {X 0,Y 379.079,Z 812.597,A -85,B 0,C 180,E1 -18406.598,E2 -18406.598} C_VEL
LIN {X 0,Y 374.178,Z 833.62,A -85,B 0,C 180,E1 -18408.595,E2 -18408.595} C_VEL
LIN {X 0,Y 369.316,Z 853.128,A -85,B 0,C 180,E1 -18410.81,E2 -18410.81} C_VEL
LIN {X 0,Y 364.284,Z 872.858,A -85,B 0,C 180,E1 -18413.443,E2 -18413.443} C_VEL
LIN {X 0,Y 359.737,Z 890.512,A -85,B 0,C 180,E1 -18416.21,E2 -18416.21} C_VEL
LIN {X 0,Y 355.626,Z 906.727,A -85,B 0,C 180,E1 -18419.222,E2 -18419.222} C_VEL
LIN {X 0,Y 352.112,Z 921.437,A -85,B 0,C 180,E1 -18422.428,E2 -18422.428} C_VEL
LIN {X 0,Y 349.518,Z 933.352,A -85,B 0,C 180,E1 -18425.493,E2 -18425.493} C_VEL
LIN {X 0,Y 347.327,Z 945.157,A -85,B 0,C 180,E1 -18429.086,E2 -18429.086} C_VEL
LIN {X 0,Y 346.043,Z 954.062,A -85,B 0,C 180,E1 -18432.338,E2 -18432.338} C_VEL
LIN {X 0,Y 345.258,Z 962.402,A -85,B 0,C 180,E1 -18436.092,E2 -18436.092} C_VEL
LIN {X 0,Y 345.051,Z 967.893,A -85,B 0,C 180,E1 -18439.222,E2 -18439.222} C_VEL
LIN {X 0,Y 345.124,Z 972.521,A -85,B 0,C 180,E1 -18442.676,E2 -18442.676} C_VEL
LIN {X 0,Y 345.329,Z 975.386,A -85,B 0,C 180,E1 -18446.015,E2 -18446.015} C_VEL
LIN {X 0,Y 345.409,Z 976.769,A -85,B 0,C 180,E1 -18449.005,E2 -18449.005} C_VEL
LIN {X 0,Y 345.305,Z 977.005,A -85,B 0,C 180,E1 -18452.157,E2 -18452.157} C_VEL
LIN {X 0,Y 345.046,Z 975.752,A -85,B 0,C 180,E1 -18455.654,E2 -18455.654} C_VEL
LIN {X 0,Y 344.799,Z 973.147,A -85,B 0,C 180,E1 -18459.009,E2 -18459.009} C_VEL
LIN {X 0,Y 344.817,Z 969.073,A -85,B 0,C 180,E1 -18462.561,E2 -18462.561} C_VEL
LIN {X 0,Y 345.466,Z 962.594,A -85,B 0,C 180,E1 -18466.651,E2 -18466.651} C_VEL
LIN {X 0,Y 346.892,Z 955.072,A -85,B 0,C 180,E1 -18470.412,E2 -18470.412} C_VEL
LIN {X 0,Y 349.593,Z 944.98,A -85,B 0,C 180,E1 -18474.502,E2 -18474.502} C_VEL
LIN {X 0,Y 353.495,Z 933.505,A -85,B 0,C 180,E1 -18478.394,E2 -18478.394} C_VEL
LIN {X 0,Y 358.699,Z 920.105,A -85,B 0,C 180,E1 -18482.169,E2 -18482.169} C_VEL
LIN {X 0,Y 365.389,Z 904.751,A -85,B 0,C 180,E1 -18485.847,E2 -18485.847} C_VEL
LIN {X 0,Y 373.195,Z 888.055,A -85,B 0,C 180,E1 -18489.221,E2 -18489.221} C_VEL
LIN {X 0,Y 381.941,Z 870.073,A -85,B 0,C 180,E1 -18492.284,E2 -18492.284} C_VEL
LIN {X 0,Y 392.294,Z 849.528,A -85,B 0,C 180,E1 -18495.223,E2 -18495.223} C_VEL
LIN {X 0,Y 402.876,Z 828.807,A -85,B 0,C 180,E1 -18497.698,E2 -18497.698} C_VEL
LIN {X 0,Y 414.345,Z 806.273,A -85,B 0,C 180,E1 -18499.905,E2 -18499.905} C_VEL
LIN {X 0,Y 425.952,Z 783.125,A -85,B 0,C 180,E1 -18501.741,E2 -18501.741} C_VEL
LIN {X 0,Y 430.183,Z 774.498,A -85,B 0,C 180,E1 -18502.337,E2 -18502.337} C_VEL
LIN {X 0,Y 417.846,Z 793.984,A -85,B 0,C 180,E1 -18504.022,E2 -18504.022} C_VEL
LIN {X 0,Y 406.069,Z 812.314,A -85,B 0,C 180,E1 -18506.016,E2 -18506.016} C_VEL
LIN {X 0,Y 394.907,Z 829.925,A -85,B 0,C 180,E1 -18508.391,E2 -18508.391} C_VEL
LIN {X 0,Y 384.787,Z 846.339,A -85,B 0,C 180,E1 -18511.097,E2 -18511.097} C_VEL
LIN {X 0,Y 376.157,Z 860.63,A -85,B 0,C 180,E1 -18513.985,E2 -18513.985} C_VEL
LIN {X 0,Y 369.175,Z 872.195,A -85,B 0,C 180,E1 -18516.876,E2 -18516.876} C_VEL
LIN {X 0,Y 363.564,Z 881.294,A -85,B 0,C 180,E1 -18519.725,E2 -18519.725} C_VEL
LIN {X 0,Y 358.867,Z 888.538,A -85,B 0,C 180,E1 -18522.655,E2 -18522.655} C_VEL
LIN {X 0,Y 355.002,Z 893.969,A -85,B 0,C 180,E1 -18525.674,E2 -18525.674} C_VEL
LIN {X 0,Y 352.008,Z 897.518,A -85,B 0,C 180,E1 -18528.697,E2 -18528.697} C_VEL
LIN {X 0,Y 349.838,Z 899.205,A -85,B 0,C 180,E1 -18531.618,E2 -18531.618} C_VEL
LIN {X 0,Y 348.25,Z 899.262,A -85,B 0,C 180,E1 -18534.563,E2 -18534.563} C_VEL
LIN {X 0,Y 347.127,Z 897.443,A -85,B 0,C 180,E1 -18537.689,E2 -18537.689} C_VEL
LIN {X 0,Y 346.52,Z 893.961,A -85,B 0,C 180,E1 -18540.661,E2 -18540.661} C_VEL
LIN {X 0,Y 346.278,Z 889.094,A -85,B 0,C 180,E1 -18543.476,E2 -18543.476} C_VEL
LIN {X 0,Y 346.374,Z 882.169,A -85,B 0,C 180,E1 -18546.464,E2 -18546.464} C_VEL
LIN {X 0,Y 346.843,Z 873.252,A -85,B 0,C 180,E1 -18549.458,E2 -18549.458} C_VEL
LIN {X 0,Y 347.693,Z 862.814,A -85,B 0,C 180,E1 -18552.287,E2 -18552.287} C_VEL
LIN {X 0,Y 349.005,Z 850.164,A -85,B 0,C 180,E1 -18555.112,E2 -18555.112} C_VEL
LIN {X 0,Y 350.714,Z 835.834,A -85,B 0,C 180,E1 -18557.779,E2 -18557.779} C_VEL
LIN {X 0,Y 352.82,Z 819.581,A -85,B 0,C 180,E1 -18560.314,E2 -18560.314} C_VEL
LIN {X 0,Y 355.155,Z 802.162,A -85,B 0,C 180,E1 -18562.592,E2 -18562.592} C_VEL
LIN {X 0,Y 357.618,Z 783.595,A -85,B 0,C 180,E1 -18564.62,E2 -18564.62} C_VEL
LIN {X 0,Y 360.204,Z 763.387,A -85,B 0,C 180,E1 -18566.458,E2 -18566.458} C_VEL
LIN {X 0,Y 362.917,Z 741.169,A -85,B 0,C 180,E1 -18568.108,E2 -18568.108} C_VEL
LIN {X 0,Y 365.401,Z 718.55,A -85,B 0,C 180,E1 -18569.453,E2 -18569.453} C_VEL
LIN {X 0,Y 367.676,Z 694.971,A -85,B 0,C 180,E1 -18570.533,E2 -18570.533} C_VEL
LIN {X 0,Y 369.734,Z 668.465,A -85,B 0,C 180,E1 -18571.406,E2 -18571.406} C_VEL
LIN {X 0,Y 381.298,Z 513.044,A -85,B 0,C 180,E1 -18575.799,E2 -18575.799} C_VEL
LIN {X 0,Y 380.562,Z 497.793,A -85,B 0,C 180,E1 -18576.427,E2 -18576.427} C_VEL
LIN {X 0,Y 381.91,Z 497.424,A -85,B 0,C 180,E1 -18576.698,E2 -18576.698} C_VEL
LIN {X 0,Y 384.062,Z 494.383,A -85,B 0,C 180,E1 -18577.041,E2 -18577.041} C_VEL
LIN {X 0,Y 387.078,Z 487.132,A -85,B 0,C 180,E1 -18577.411,E2 -18577.411} C_VEL
LIN {X 0,Y 389.611,Z 478.921,A -85,B 0,C 180,E1 -18577.648,E2 -18577.648} C_VEL
LIN {X 0,Y 392.602,Z 474.92,A -85,B 0,C 180,E1 -18578.107,E2 -18578.107} C_VEL
LIN {X 0,Y 395.882,Z 467.794,A -85,B 0,C 180,E1 -18578.517,E2 -18578.517} C_VEL
LIN {X 0,Y 399.162,Z 458.109,A -85,B 0,C 180,E1 -18578.843,E2 -18578.843} C_VEL
LIN {X 0,Y 402.818,Z 452.307,A -85,B 0,C 180,E1 -18579.339,E2 -18579.339} C_VEL
LIN {X 0,Y 405.644,Z 446.453,A -85,B 0,C 180,E1 -18579.674,E2 -18579.674} C_VEL
LIN {X 0,Y 410.988,Z 441.796,A -85,B 0,C 180,E1 -18580.465,E2 -18580.465} C_VEL
LIN {X 0,Y 414.182,Z 438.511,A -85,B 0,C 180,E1 -18580.907,E2 -18580.907} C_VEL
LIN {X 0,Y 418.775,Z 435.159,A -85,B 0,C 180,E1 -18581.561,E2 -18581.561} C_VEL
LIN {X 0,Y 414.552,Z 502.765,A -85,B 0,C 180,E1 -18582.771,E2 -18582.771} C_VEL
LIN {X 0,Y 409.675,Z 559.247,A -85,B 0,C 180,E1 -18583.995,E2 -18583.995} C_VEL
LIN {X 0,Y 403.386,Z 618.02,A -85,B 0,C 180,E1 -18585.503,E2 -18585.503} C_VEL
LIN {X 0,Y 398.632,Z 661.485,A -85,B 0,C 180,E1 -18586.862,E2 -18586.862} C_VEL
LIN {X 0,Y 395.816,Z 689.205,A -85,B 0,C 180,E1 -18587.928,E2 -18587.928} C_VEL
LIN {X 0,Y 393.023,Z 709.908,A -85,B 0,C 180,E1 -18588.976,E2 -18588.976} C_VEL
LIN {X 0,Y 389.526,Z 730.303,A -85,B 0,C 180,E1 -18590.27,E2 -18590.27} C_VEL
LIN {X 0,Y 385.519,Z 749.859,A -85,B 0,C 180,E1 -18591.801,E2 -18591.801} C_VEL
LIN {X 0,Y 380.981,Z 768.959,A -85,B 0,C 180,E1 -18593.62,E2 -18593.62} C_VEL
LIN {X 0,Y 376.142,Z 787.06,A -85,B 0,C 180,E1 -18595.698,E2 -18595.698} C_VEL
LIN {X 0,Y 371.346,Z 803.534,A -85,B 0,C 180,E1 -18597.964,E2 -18597.964} C_VEL
LIN {X 0,Y 366.423,Z 819.368,A -85,B 0,C 180,E1 -18600.582,E2 -18600.582} C_VEL
LIN {X 0,Y 361.821,Z 833.553,A -85,B 0,C 180,E1 -18603.405,E2 -18603.405} C_VEL
LIN {X 0,Y 357.662,Z 846.148,A -85,B 0,C 180,E1 -18606.436,E2 -18606.436} C_VEL
LIN {X 0,Y 354.056,Z 857.156,A -85,B 0,C 180,E1 -18609.674,E2 -18609.674} C_VEL
LIN {X 0,Y 351.093,Z 866.569,A -85,B 0,C 180,E1 -18613.119,E2 -18613.119} C_VEL
LIN {X 0,Y 348.93,Z 873.941,A -85,B 0,C 180,E1 -18616.578,E2 -18616.578} C_VEL
LIN {X 0,Y 347.453,Z 879.498,A -85,B 0,C 180,E1 -18620.057,E2 -18620.057} C_VEL
LIN {X 0,Y 346.57,Z 883.344,A -85,B 0,C 180,E1 -18623.539,E2 -18623.539} C_VEL
LIN {X 0,Y 346.126,Z 885.557,A -85,B 0,C 180,E1 -18627.019,E2 -18627.019} C_VEL
LIN {X 0,Y 346.019,Z 886.198,A -85,B 0,C 180,E1 -18630.331,E2 -18630.331} C_VEL
LIN {X 0,Y 346.194,Z 885.284,A -85,B 0,C 180,E1 -18633.809,E2 -18633.809} C_VEL
LIN {X 0,Y 346.722,Z 882.699,A -85,B 0,C 180,E1 -18637.29,E2 -18637.29} C_VEL
LIN {X 0,Y 346.846,Z 882.204,A -85,B 0,C 180,E1 -18637.815,E2 -18637.815} C_VEL
LIN {X 0,Y 346.156,Z 880.919,A -85,B 0,C 180,E1 -18639.074,E2 -18639.074} C_VEL
LIN {X 0,Y 341.298,Z 877.302,A -85,B 0,C 180,E1 -18642.377,E2 -18642.377} C_VEL
LIN {X 0,Y 341.041,Z 875.505,A -85,B 0,C 180,E1 -18643.555,E2 -18643.555} C_VEL
LIN {X 0,Y 343.368,Z 867.961,A -85,B 0,C 180,E1 -18647.226,E2 -18647.226} C_VEL
LIN {X 0,Y 346.501,Z 858.52,A -85,B 0,C 180,E1 -18650.79,E2 -18650.79} C_VEL
LIN {X 0,Y 350.265,Z 847.584,A -85,B 0,C 180,E1 -18654.093,E2 -18654.093} C_VEL
LIN {X 0,Y 354.598,Z 835.063,A -85,B 0,C 180,E1 -18657.181,E2 -18657.181} C_VEL
LIN {X 0,Y 359.499,Z 820.631,A -85,B 0,C 180,E1 -18660.117,E2 -18660.117} C_VEL
LIN {X 0,Y 364.654,Z 804.731,A -85,B 0,C 180,E1 -18662.789,E2 -18662.789} C_VEL
LIN {X 0,Y 369.81,Z 787.687,A -85,B 0,C 180,E1 -18665.163,E2 -18665.163} C_VEL
LIN {X 0,Y 374.841,Z 769.486,A -85,B 0,C 180,E1 -18667.266,E2 -18667.266} C_VEL
LIN {X 0,Y 379.577,Z 750.118,A -85,B 0,C 180,E1 -18669.116,E2 -18669.116} C_VEL
LIN {X 0,Y 383.71,Z 730.552,A -85,B 0,C 180,E1 -18670.652,E2 -18670.652} C_VEL
LIN {X 0,Y 387.39,Z 709.552,A -85,B 0,C 180,E1 -18671.982,E2 -18671.982} C_VEL
LIN {X 0,Y 390.342,Z 687.798,A -85,B 0,C 180,E1 -18673.064,E2 -18673.064} C_VEL
LIN {X 0,Y 394.08,Z 651.812,A -85,B 0,C 180,E1 -18674.395,E2 -18674.395} C_VEL
LIN {X 0,Y 399.63,Z 604.047,A -85,B 0,C 180,E1 -18675.817,E2 -18675.817} C_VEL
LIN {X 0,Y 405.331,Z 550.107,A -85,B 0,C 180,E1 -18677.161,E2 -18677.161} C_VEL
LIN {X 0,Y 410.073,Z 493.875,A -85,B 0,C 180,E1 -18678.348,E2 -18678.348} C_VEL
LIN {X 0,Y 414.662,Z 421.018,A -85,B 0,C 180,E1 -18679.639,E2 -18679.639} C_VEL
LIN {X 0,Y 422.447,Z 386.912,A -85,B 0,C 180,E1 -18680.848,E2 -18680.848} C_VEL
LIN {X 0,Y 416.547,Z 369.52,A -85,B 0,C 180,E1 -18683.527,E2 -18683.527} C_VEL
LIN {X 0,Y 410.555,Z 353.951,A -85,B 0,C 180,E1 -18686.269,E2 -18686.269} C_VEL
LIN {X 0,Y 403.937,Z 338.684,A -85,B 0,C 180,E1 -18689.341,E2 -18689.341} C_VEL
LIN {X 0,Y 397.815,Z 326.026,A -85,B 0,C 180,E1 -18692.29,E2 -18692.29} C_VEL
LIN {X 0,Y 391.735,Z 314.733,A -85,B 0,C 180,E1 -18695.374,E2 -18695.374} C_VEL
LIN {X 0,Y 387.346,Z 307.149,A -85,B 0,C 180,E1 -18697.779,E2 -18697.779} C_VEL
LIN {X 0,Y 384.831,Z 302.805,A -85,B 0,C 180,E1 -18699.307,E2 -18699.307} C_VEL
LIN {X 0,Y 381.89,Z 298.168,A -85,B 0,C 180,E1 -18701.055,E2 -18701.055} C_VEL
LIN {X 0,Y 378.815,Z 293.128,A -85,B 0,C 180,E1 -18703.2,E2 -18703.2} C_VEL
LIN {X 0,Y 376.044,Z 288.933,A -85,B 0,C 180,E1 -18705.211,E2 -18705.211} C_VEL
LIN {X 0,Y 375.141,Z 287.663,A -85,B 0,C 180,E1 -18705.963,E2 -18705.963} C_VEL
LIN {X 0,Y 372.535,Z 283.918,A -85,B 0,C 180,E1 -18708.23,E2 -18708.23} C_VEL
LIN {X 0,Y 371.837,Z 282.354,A -85,B 0,C 180,E1 -18708.993,E2 -18708.993} C_VEL
LIN {X 0,Y 369.033,Z 279.335,A -85,B 0,C 180,E1 -18712.057,E2 -18712.057} C_VEL
LIN {X 0,Y 367.973,Z 276.423,A -85,B 0,C 180,E1 -18713.917,E2 -18713.917} C_VEL
LIN {X 0,Y 365.363,Z 274.251,A -85,B 0,C 180,E1 -18721.255,E2 -18721.255} C_VEL
LIN {X 0,Y 366.194,Z 274.958,A -85,B 0,C 180,E1 -18725.798,E2 -18725.798} C_VEL
LIN {X 0,Y 368.615,Z 276.787,A -85,B 0,C 180,E1 -18729.919,E2 -18729.919} C_VEL
LIN {X 0,Y 369.762,Z 283.067,A -85,B 0,C 180,E1 -18732.295,E2 -18732.295} C_VEL
LIN {X 0,Y 372.082,Z 292.23,A -85,B 0,C 180,E1 -18735.349,E2 -18735.349} C_VEL
LIN {X 0,Y 376.983,Z 307.006,A -85,B 0,C 180,E1 -18739.645,E2 -18739.645} C_VEL
LIN {X 0,Y 384.709,Z 326.553,A -85,B 0,C 180,E1 -18744.369,E2 -18744.369} C_VEL
LIN {X 0,Y 391.347,Z 341.571,A -85,B 0,C 180,E1 -18747.484,E2 -18747.484} C_VEL
LIN {X 0,Y 393.247,Z 345.859,A -85,B 0,C 180,E1 -18748.204,E2 -18748.204} C_VEL
LIN {X 0,Y 412.614,Z 375.965,A -85,B 0,C 180,E1 -18751.749,E2 -18751.749} C_VEL
LIN {X 0,Y 417.438,Z 384.037,A -85,B 0,C 180,E1 -18752.59,E2 -18752.59} C_VEL
LIN {X 0,Y 395.572,Z 650.308,A -85,B 0,C 180,E1 -18758.52,E2 -18758.52} C_VEL
LIN {X 0,Y 392.035,Z 694.97,A -85,B 0,C 180,E1 -18759.595,E2 -18759.595} C_VEL
LIN {X 0,Y 389.157,Z 718.638,A -85,B 0,C 180,E1 -18760.377,E2 -18760.377} C_VEL
LIN {X 0,Y 385.477,Z 743.215,A -85,B 0,C 180,E1 -18761.441,E2 -18761.441} C_VEL
LIN {X 0,Y 381.496,Z 766.089,A -85,B 0,C 180,E1 -18762.677,E2 -18762.677} C_VEL
LIN {X 0,Y 377.045,Z 788.248,A -85,B 0,C 180,E1 -18764.165,E2 -18764.165} C_VEL
LIN {X 0,Y 371.839,Z 811.835,A -85,B 0,C 180,E1 -18766.071,E2 -18766.071} C_VEL
LIN {X 0,Y 366.828,Z 832.877,A -85,B 0,C 180,E1 -18768.101,E2 -18768.101} C_VEL
LIN {X 0,Y 361.884,Z 852.27,A -85,B 0,C 180,E1 -18770.338,E2 -18770.338} C_VEL
LIN {X 0,Y 356.722,Z 872.11,A -85,B 0,C 180,E1 -18773.021,E2 -18773.021} C_VEL
LIN {X 0,Y 352.014,Z 889.979,A -85,B 0,C 180,E1 -18775.875,E2 -18775.875} C_VEL
LIN {X 0,Y 347.3,Z 908.742,A -85,B 0,C 180,E1 -18779.364,E2 -18779.364} C_VEL
LIN {X 0,Y 344.138,Z 921.897,A -85,B 0,C 180,E1 -18782.298,E2 -18782.298} C_VEL
LIN {X 0,Y 341.349,Z 934.307,A -85,B 0,C 180,E1 -18785.643,E2 -18785.643} C_VEL
LIN {X 0,Y 339.31,Z 944.889,A -85,B 0,C 180,E1 -18789.111,E2 -18789.111} C_VEL
LIN {X 0,Y 337.85,Z 955.285,A -85,B 0,C 180,E1 -18793.14,E2 -18793.14} C_VEL
LIN {X 0,Y 337.264,Z 962.477,A -85,B 0,C 180,E1 -18796.63,E2 -18796.63} C_VEL
LIN {X 0,Y 337.127,Z 968.432,A -85,B 0,C 180,E1 -18800.267,E2 -18800.267} C_VEL
LIN {X 0,Y 337.281,Z 972.371,A -85,B 0,C 180,E1 -18803.703,E2 -18803.703} C_VEL
LIN {X 0,Y 337.444,Z 974.7,A -85,B 0,C 180,E1 -18806.773,E2 -18806.773} C_VEL
LIN {X 0,Y 337.483,Z 975.907,A -85,B 0,C 180,E1 -18810,E2 -18810} C_VEL
LIN {X 0,Y 337.293,Z 975.724,A -85,B 0,C 180,E1 -18813.399,E2 -18813.399} C_VEL
LIN {X 0,Y 336.994,Z 974.236,A -85,B 0,C 180,E1 -18816.645,E2 -18816.645} C_VEL
LIN {X 0,Y 336.797,Z 971.576,A -85,B 0,C 180,E1 -18819.915,E2 -18819.915} C_VEL
LIN {X 0,Y 336.949,Z 966.726,A -85,B 0,C 180,E1 -18823.982,E2 -18823.982} C_VEL
LIN {X 0,Y 337.782,Z 960.62,A -85,B 0,C 180,E1 -18827.752,E2 -18827.752} C_VEL
LIN {X 0,Y 339.63,Z 952.598,A -85,B 0,C 180,E1 -18831.774,E2 -18831.774} C_VEL
LIN {X 0,Y 342.657,Z 942.693,A -85,B 0,C 180,E1 -18835.772,E2 -18835.772} C_VEL
LIN {X 0,Y 347.253,Z 930.62,A -85,B 0,C 180,E1 -18839.877,E2 -18839.877} C_VEL
LIN {X 0,Y 353.116,Z 917.09,A -85,B 0,C 180,E1 -18843.711,E2 -18843.711} C_VEL
LIN {X 0,Y 360.941,Z 900.734,A -85,B 0,C 180,E1 -18847.6,E2 -18847.6} C_VEL
LIN {X 0,Y 369.877,Z 883.356,A -85,B 0,C 180,E1 -18851.064,E2 -18851.064} C_VEL
LIN {X 0,Y 380.006,Z 864.49,A -85,B 0,C 180,E1 -18854.209,E2 -18854.209} C_VEL
LIN {X 0,Y 391.274,Z 843.862,A -85,B 0,C 180,E1 -18857.067,E2 -18857.067} C_VEL
LIN {X 0,Y 403.382,Z 822.083,A -85,B 0,C 180,E1 -18859.551,E2 -18859.551} C_VEL
LIN {X 0,Y 415.815,Z 799.709,A -85,B 0,C 180,E1 -18861.621,E2 -18861.621} C_VEL
LIN {X 0,Y 421.054,Z 790.222,A -85,B 0,C 180,E1 -18862.388,E2 -18862.388} C_VEL
LIN {X 0,Y 408.407,Z 808.115,A -85,B 0,C 180,E1 -18864.187,E2 -18864.187} C_VEL
LIN {X 0,Y 395.922,Z 825.807,A -85,B 0,C 180,E1 -18866.421,E2 -18866.421} C_VEL
LIN {X 0,Y 384.504,Z 842.367,A -85,B 0,C 180,E1 -18869.01,E2 -18869.01} C_VEL
LIN {X 0,Y 374.661,Z 856.99,A -85,B 0,C 180,E1 -18871.811,E2 -18871.811} C_VEL
LIN {X 0,Y 366.267,Z 869.642,A -85,B 0,C 180,E1 -18874.794,E2 -18874.794} C_VEL
LIN {X 0,Y 359.178,Z 880.187,A -85,B 0,C 180,E1 -18877.925,E2 -18877.925} C_VEL
LIN {X 0,Y 353.543,Z 888.234,A -85,B 0,C 180,E1 -18881.02,E2 -18881.02} C_VEL
LIN {X 0,Y 348.923,Z 894.302,A -85,B 0,C 180,E1 -18884.203,E2 -18884.203} C_VEL
LIN {X 0,Y 345.265,Z 898.383,A -85,B 0,C 180,E1 -18887.455,E2 -18887.455} C_VEL
LIN {X 0,Y 342.501,Z 900.474,A -85,B 0,C 180,E1 -18890.76,E2 -18890.76} C_VEL
LIN {X 0,Y 340.605,Z 900.563,A -85,B 0,C 180,E1 -18893.933,E2 -18893.933} C_VEL
LIN {X 0,Y 339.39,Z 898.942,A -85,B 0,C 180,E1 -18896.96,E2 -18896.96} C_VEL
LIN {X 0,Y 338.659,Z 895.626,A -85,B 0,C 180,E1 -18900,E2 -18900} C_VEL
LIN {X 0,Y 338.323,Z 890.618,A -85,B 0,C 180,E1 -18903.049,E2 -18903.049} C_VEL
LIN {X 0,Y 338.355,Z 884.258,A -85,B 0,C 180,E1 -18905.937,E2 -18905.937} C_VEL
LIN {X 0,Y 338.728,Z 876.113,A -85,B 0,C 180,E1 -18908.83,E2 -18908.83} C_VEL
LIN {X 0,Y 339.498,Z 866.06,A -85,B 0,C 180,E1 -18911.725,E2 -18911.725} C_VEL
LIN {X 0,Y 340.735,Z 853.868,A -85,B 0,C 180,E1 -18914.618,E2 -18914.618} C_VEL
LIN {X 0,Y 342.364,Z 840.096,A -85,B 0,C 180,E1 -18917.331,E2 -18917.331} C_VEL
LIN {X 0,Y 344.487,Z 823.708,A -85,B 0,C 180,E1 -18920.029,E2 -18920.029} C_VEL
LIN {X 0,Y 346.888,Z 806.117,A -85,B 0,C 180,E1 -18922.453,E2 -18922.453} C_VEL
LIN {X 0,Y 349.557,Z 786.744,A -85,B 0,C 180,E1 -18924.685,E2 -18924.685} C_VEL
LIN {X 0,Y 352.282,Z 766.215,A -85,B 0,C 180,E1 -18926.645,E2 -18926.645} C_VEL
LIN {X 0,Y 354.894,Z 745.696,A -85,B 0,C 180,E1 -18928.251,E2 -18928.251} C_VEL
LIN {X 0,Y 357.48,Z 723.115,A -85,B 0,C 180,E1 -18929.675,E2 -18929.675} C_VEL
LIN {X 0,Y 359.936,Z 699.006,A -85,B 0,C 180,E1 -18930.856,E2 -18930.856} C_VEL
LIN {X 0,Y 361.994,Z 674.681,A -85,B 0,C 180,E1 -18931.731,E2 -18931.731} C_VEL
LIN {X 0,Y 373.543,Z 526.866,A -85,B 0,C 180,E1 -18936.031,E2 -18936.031} C_VEL
LIN {X 0,Y 374.749,Z 526.346,A -85,B 0,C 180,E1 -18936.275,E2 -18936.275} C_VEL
LIN {X 0,Y 377.145,Z 522.135,A -85,B 0,C 180,E1 -18936.621,E2 -18936.621} C_VEL
LIN {X 0,Y 382.359,Z 508.589,A -85,B 0,C 180,E1 -18937.198,E2 -18937.198} C_VEL
LIN {X 0,Y 383.808,Z 503.98,A -85,B 0,C 180,E1 -18937.327,E2 -18937.327} C_VEL
LIN {X 0,Y 386.767,Z 500.125,A -85,B 0,C 180,E1 -18937.786,E2 -18937.786} C_VEL
LIN {X 0,Y 390.129,Z 493.051,A -85,B 0,C 180,E1 -18938.205,E2 -18938.205} C_VEL
LIN {X 0,Y 393.434,Z 483.485,A -85,B 0,C 180,E1 -18938.534,E2 -18938.534} C_VEL
LIN {X 0,Y 397.09,Z 477.73,A -85,B 0,C 180,E1 -18939.038,E2 -18939.038} C_VEL
LIN {X 0,Y 400.819,Z 469.022,A -85,B 0,C 180,E1 -18939.458,E2 -18939.458} C_VEL
LIN {X 0,Y 403.182,Z 462.32,A -85,B 0,C 180,E1 -18939.688,E2 -18939.688} C_VEL
LIN {X 0,Y 407.332,Z 455.185,A -85,B 0,C 180,E1 -18940.211,E2 -18940.211} C_VEL
LIN {X 0,Y 408.702,Z 452.461,A -85,B 0,C 180,E1 -18940.37,E2 -18940.37} C_VEL
LIN {X 0,Y 412.767,Z 449.062,A -85,B 0,C 180,E1 -18940.957,E2 -18940.957} C_VEL
LIN {X 0,Y 408.905,Z 507.719,A -85,B 0,C 180,E1 -18942.03,E2 -18942.03} C_VEL
LIN {X 0,Y 403.966,Z 562.831,A -85,B 0,C 180,E1 -18943.241,E2 -18943.241} C_VEL
LIN {X 0,Y 397.6,Z 620.328,A -85,B 0,C 180,E1 -18944.737,E2 -18944.737} C_VEL
LIN {X 0,Y 392.747,Z 663.489,A -85,B 0,C 180,E1 -18946.111,E2 -18946.111} C_VEL
LIN {X 0,Y 389.778,Z 691.389,A -85,B 0,C 180,E1 -18947.206,E2 -18947.206} C_VEL
LIN {X 0,Y 386.8,Z 712.442,A -85,B 0,C 180,E1 -18948.297,E2 -18948.297} C_VEL
LIN {X 0,Y 383.19,Z 732.554,A -85,B 0,C 180,E1 -18949.604,E2 -18949.604} C_VEL
LIN {X 0,Y 379.142,Z 751.575,A -85,B 0,C 180,E1 -18951.122,E2 -18951.122} C_VEL
LIN {X 0,Y 374.611,Z 769.999,A -85,B 0,C 180,E1 -18952.899,E2 -18952.899} C_VEL
LIN {X 0,Y 369.599,Z 788.112,A -85,B 0,C 180,E1 -18955.003,E2 -18955.003} C_VEL
LIN {X 0,Y 364.456,Z 805.095,A -85,B 0,C 180,E1 -18957.38,E2 -18957.38} C_VEL
LIN {X 0,Y 359.5,Z 820.419,A -85,B 0,C 180,E1 -18959.957,E2 -18959.957} C_VEL
LIN {X 0,Y 354.702,Z 834.6,A -85,B 0,C 180,E1 -18962.827,E2 -18962.827} C_VEL
LIN {X 0,Y 350.244,Z 847.507,A -85,B 0,C 180,E1 -18966.001,E2 -18966.001} C_VEL
LIN {X 0,Y 346.406,Z 858.676,A -85,B 0,C 180,E1 -18969.381,E2 -18969.381} C_VEL
LIN {X 0,Y 343.335,Z 867.971,A -85,B 0,C 180,E1 -18972.894,E2 -18972.894} C_VEL
LIN {X 0,Y 341.086,Z 875.281,A -85,B 0,C 180,E1 -18976.437,E2 -18976.437} C_VEL
LIN {X 0,Y 339.498,Z 880.979,A -85,B 0,C 180,E1 -18980.164,E2 -18980.164} C_VEL
LIN {X 0,Y 338.608,Z 884.646,A -85,B 0,C 180,E1 -18983.727,E2 -18983.727} C_VEL
LIN {X 0,Y 338.183,Z 886.622,A -85,B 0,C 180,E1 -18987.119,E2 -18987.119} C_VEL
LIN {X 0,Y 338.077,Z 887.155,A -85,B 0,C 180,E1 -18990.678,E2 -18990.678} C_VEL
LIN {X 0,Y 338.287,Z 886.201,A -85,B 0,C 180,E1 -18994.068,E2 -18994.068} C_VEL
LIN {X 0,Y 338.874,Z 883.559,A -85,B 0,C 180,E1 -18997.63,E2 -18997.63} C_VEL
LIN {X 0,Y 339.952,Z 879.257,A -85,B 0,C 180,E1 -19001.193,E2 -19001.193} C_VEL
LIN {X 0,Y 341.041,Z 875.505,A -85,B 0,C 180,E1 -19003.555,E2 -19003.555} C_VEL
LIN {X 0,Y 340.777,Z 873.444,A -85,B 0,C 180,E1 -19004.811,E2 -19004.811} C_VEL
LIN {X 0,Y 336.924,Z 867.433,A -85,B 0,C 180,E1 -19008.197,E2 -19008.197} C_VEL
LIN {X 0,Y 337.099,Z 865.021,A -85,B 0,C 180,E1 -19009.257,E2 -19009.257} C_VEL
LIN {X 0,Y 340.514,Z 855.39,A -85,B 0,C 180,E1 -19012.623,E2 -19012.623} C_VEL
LIN {X 0,Y 344.323,Z 844.841,A -85,B 0,C 180,E1 -19015.638,E2 -19015.638} C_VEL
LIN {X 0,Y 348.823,Z 832.357,A -85,B 0,C 180,E1 -19018.6,E2 -19018.6} C_VEL
LIN {X 0,Y 353.805,Z 818.12,A -85,B 0,C 180,E1 -19021.407,E2 -19021.407} C_VEL
LIN {X 0,Y 359.142,Z 802.082,A -85,B 0,C 180,E1 -19024.029,E2 -19024.029} C_VEL
LIN {X 0,Y 364.411,Z 784.985,A -85,B 0,C 180,E1 -19026.347,E2 -19026.347} C_VEL
LIN {X 0,Y 369.446,Z 766.967,A -85,B 0,C 180,E1 -19028.377,E2 -19028.377} C_VEL
LIN {X 0,Y 374.158,Z 747.889,A -85,B 0,C 180,E1 -19030.155,E2 -19030.155} C_VEL
LIN {X 0,Y 378.247,Z 728.625,A -85,B 0,C 180,E1 -19031.631,E2 -19031.631} C_VEL
LIN {X 0,Y 381.733,Z 708.857,A -85,B 0,C 180,E1 -19032.864,E2 -19032.864} C_VEL
LIN {X 0,Y 384.554,Z 688.472,A -85,B 0,C 180,E1 -19033.876,E2 -19033.876} C_VEL
LIN {X 0,Y 388.931,Z 648.613,A -85,B 0,C 180,E1 -19035.356,E2 -19035.356} C_VEL
LIN {X 0,Y 394.759,Z 599.861,A -85,B 0,C 180,E1 -19036.79,E2 -19036.79} C_VEL
LIN {X 0,Y 400.823,Z 542.636,A -85,B 0,C 180,E1 -19038.195,E2 -19038.195} C_VEL
LIN {X 0,Y 405.2,Z 490.011,A -85,B 0,C 180,E1 -19039.284,E2 -19039.284} C_VEL
LIN {X 0,Y 409.427,Z 423.831,A -85,B 0,C 180,E1 -19040.454,E2 -19040.454} C_VEL
LIN {X 0,Y 417.121,Z 390.364,A -85,B 0,C 180,E1 -19041.621,E2 -19041.621} C_VEL
LIN {X 0,Y 411.349,Z 373.311,A -85,B 0,C 180,E1 -19044.311,E2 -19044.311} C_VEL
LIN {X 0,Y 405.097,Z 356.95,A -85,B 0,C 180,E1 -19047.279,E2 -19047.279} C_VEL
LIN {X 0,Y 398.971,Z 342.808,A -85,B 0,C 180,E1 -19050.249,E2 -19050.249} C_VEL
LIN {X 0,Y 393.349,Z 331.094,A -85,B 0,C 180,E1 -19053.097,E2 -19053.097} C_VEL
LIN {X 0,Y 387.688,Z 320.219,A -85,B 0,C 180,E1 -19056.114,E2 -19056.114} C_VEL
LIN {X 0,Y 382.254,Z 310.598,A -85,B 0,C 180,E1 -19059.321,E2 -19059.321} C_VEL
LIN {X 0,Y 378.856,Z 305.168,A -85,B 0,C 180,E1 -19061.456,E2 -19061.456} C_VEL
LIN {X 0,Y 376.111,Z 300.461,A -85,B 0,C 180,E1 -19063.473,E2 -19063.473} C_VEL
LIN {X 0,Y 373.364,Z 296.078,A -85,B 0,C 180,E1 -19065.578,E2 -19065.578} C_VEL
LIN {X 0,Y 370.31,Z 291.589,A -85,B 0,C 180,E1 -19068.395,E2 -19068.395} C_VEL
LIN {X 0,Y 369.546,Z 289.935,A -85,B 0,C 180,E1 -19069.24,E2 -19069.24} C_VEL
LIN {X 0,Y 366.73,Z 286.813,A -85,B 0,C 180,E1 -19072.322,E2 -19072.322} C_VEL
LIN {X 0,Y 365.789,Z 284.091,A -85,B 0,C 180,E1 -19074.195,E2 -19074.195} C_VEL
LIN {X 0,Y 363.563,Z 282.033,A -85,B 0,C 180,E1 -19081.418,E2 -19081.418} C_VEL
LIN {X 0,Y 364.542,Z 282.885,A -85,B 0,C 180,E1 -19086.141,E2 -19086.141} C_VEL
LIN {X 0,Y 366.736,Z 284.467,A -85,B 0,C 180,E1 -19089.653,E2 -19089.653} C_VEL
LIN {X 0,Y 367.714,Z 290.381,A -85,B 0,C 180,E1 -19091.887,E2 -19091.887} C_VEL
LIN {X 0,Y 369.906,Z 299.664,A -85,B 0,C 180,E1 -19095,E2 -19095} C_VEL
LIN {X 0,Y 374.555,Z 313.976,A -85,B 0,C 180,E1 -19099.169,E2 -19099.169} C_VEL
LIN {X 0,Y 381.95,Z 333.396,A -85,B 0,C 180,E1 -19103.898,E2 -19103.898} C_VEL
LIN {X 0,Y 388.176,Z 347.845,A -85,B 0,C 180,E1 -19106.918,E2 -19106.918} C_VEL
LIN {X 0,Y 391.642,Z 356.438,A -85,B 0,C 180,E1 -19108.372,E2 -19108.372} C_VEL
LIN {X 0,Y 408.949,Z 383.589,A -85,B 0,C 180,E1 -19111.55,E2 -19111.55} C_VEL
LIN {X 0,Y 411.089,Z 387.345,A -85,B 0,C 180,E1 -19111.936,E2 -19111.936} C_VEL
LIN {X 0,Y 388.3,Z 656.144,A -85,B 0,C 180,E1 -19118.047,E2 -19118.047} C_VEL
LIN {X 0,Y 385.05,Z 695.395,A -85,B 0,C 180,E1 -19119.02,E2 -19119.02} C_VEL
LIN {X 0,Y 382.056,Z 719.294,A -85,B 0,C 180,E1 -19119.829,E2 -19119.829} C_VEL
LIN {X 0,Y 378.337,Z 743.436,A -85,B 0,C 180,E1 -19120.9,E2 -19120.9} C_VEL
LIN {X 0,Y 374.217,Z 766.461,A -85,B 0,C 180,E1 -19122.174,E2 -19122.174} C_VEL
LIN {X 0,Y 369.521,Z 789.281,A -85,B 0,C 180,E1 -19123.741,E2 -19123.741} C_VEL
LIN {X 0,Y 364.429,Z 811.762,A -85,B 0,C 180,E1 -19125.601,E2 -19125.601} C_VEL
LIN {X 0,Y 359.316,Z 832.761,A -85,B 0,C 180,E1 -19127.668,E2 -19127.668} C_VEL
LIN {X 0,Y 354.097,Z 852.805,A -85,B 0,C 180,E1 -19130.028,E2 -19130.028} C_VEL
LIN {X 0,Y 346.781,Z 881.406,A -85,B 0,C 180,E1 -19133.97,E2 -19133.97} C_VEL
LIN {X 0,Y 342.86,Z 896.81,A -85,B 0,C 180,E1 -19136.552,E2 -19136.552} C_VEL
LIN {X 0,Y 338.998,Z 911.599,A -85,B 0,C 180,E1 -19139.514,E2 -19139.514} C_VEL
LIN {X 0,Y 335.686,Z 924.838,A -85,B 0,C 180,E1 -19142.696,E2 -19142.696} C_VEL
LIN {X 0,Y 332.982,Z 936.48,A -85,B 0,C 180,E1 -19146.085,E2 -19146.085} C_VEL
LIN {X 0,Y 331.021,Z 946.585,A -85,B 0,C 180,E1 -19149.673,E2 -19149.673} C_VEL
LIN {X 0,Y 329.819,Z 955.151,A -85,B 0,C 180,E1 -19153.443,E2 -19153.443} C_VEL
LIN {X 0,Y 329.294,Z 962.307,A -85,B 0,C 180,E1 -19157.087,E2 -19157.087} C_VEL
LIN {X 0,Y 329.222,Z 968.117,A -85,B 0,C 180,E1 -19160.913,E2 -19160.913} C_VEL
LIN {X 0,Y 329.397,Z 971.698,A -85,B 0,C 180,E1 -19164.251,E2 -19164.251} C_VEL
LIN {X 0,Y 329.533,Z 973.873,A -85,B 0,C 180,E1 -19167.391,E2 -19167.391} C_VEL
LIN {X 0,Y 329.516,Z 974.904,A -85,B 0,C 180,E1 -19170.869,E2 -19170.869} C_VEL
LIN {X 0,Y 329.284,Z 974.461,A -85,B 0,C 180,E1 -19174.179,E2 -19174.179} C_VEL
LIN {X 0,Y 328.974,Z 972.922,A -85,B 0,C 180,E1 -19177.334,E2 -19177.334} C_VEL
LIN {X 0,Y 328.789,Z 970.053,A -85,B 0,C 180,E1 -19180.799,E2 -19180.799} C_VEL
LIN {X 0,Y 329.104,Z 965.009,A -85,B 0,C 180,E1 -19184.966,E2 -19184.966} C_VEL
LIN {X 0,Y 330.194,Z 958.667,A -85,B 0,C 180,E1 -19188.906,E2 -19188.906} C_VEL
LIN {X 0,Y 332.774,Z 949.221,A -85,B 0,C 180,E1 -19193.555,E2 -19193.555} C_VEL
LIN {X 0,Y 336.528,Z 938.905,A -85,B 0,C 180,E1 -19197.697,E2 -19197.697} C_VEL
LIN {X 0,Y 342.051,Z 926.084,A -85,B 0,C 180,E1 -19201.945,E2 -19201.945} C_VEL
LIN {X 0,Y 349.14,Z 911.666,A -85,B 0,C 180,E1 -19205.951,E2 -19205.951} C_VEL
LIN {X 0,Y 357.559,Z 895.887,A -85,B 0,C 180,E1 -19209.612,E2 -19209.612} C_VEL
LIN {X 0,Y 367.552,Z 878.113,A -85,B 0,C 180,E1 -19213.065,E2 -19213.065} C_VEL
LIN {X 0,Y 379.193,Z 858.346,A -85,B 0,C 180,E1 -19216.262,E2 -19216.262} C_VEL
LIN {X 0,Y 391.474,Z 838.016,A -85,B 0,C 180,E1 -19218.972,E2 -19218.972} C_VEL
LIN {X 0,Y 403.978,Z 817.307,A -85,B 0,C 180,E1 -19221.23,E2 -19221.23} C_VEL
LIN {X 0,Y 411.753,Z 804.434,A -85,B 0,C 180,E1 -19222.445,E2 -19222.445} C_VEL
LIN {X 0,Y 398.634,Z 821.4,A -85,B 0,C 180,E1 -19224.414,E2 -19224.414} C_VEL
LIN {X 0,Y 385.793,Z 838.082,A -85,B 0,C 180,E1 -19226.848,E2 -19226.848} C_VEL
LIN {X 0,Y 374.09,Z 853.588,A -85,B 0,C 180,E1 -19229.657,E2 -19229.657} C_VEL
LIN {X 0,Y 364.083,Z 867.125,A -85,B 0,C 180,E1 -19232.701,E2 -19232.701} C_VEL
LIN {X 0,Y 355.97,Z 878.109,A -85,B 0,C 180,E1 -19235.789,E2 -19235.789} C_VEL
LIN {X 0,Y 349.411,Z 886.787,A -85,B 0,C 180,E1 -19238.891,E2 -19238.891} C_VEL
LIN {X 0,Y 344.031,Z 893.466,A -85,B 0,C 180,E1 -19242.056,E2 -19242.056} C_VEL
LIN {X 0,Y 339.839,Z 898.112,A -85,B 0,C 180,E1 -19245.169,E2 -19245.169} C_VEL
LIN {X 0,Y 336.371,Z 901.078,A -85,B 0,C 180,E1 -19248.512,E2 -19248.512} C_VEL
LIN {X 0,Y 333.814,Z 902.079,A -85,B 0,C 180,E1 -19251.907,E2 -19251.907} C_VEL
LIN {X 0,Y 332.101,Z 901.142,A -85,B 0,C 180,E1 -19255.164,E2 -19255.164} C_VEL
LIN {X 0,Y 331.064,Z 898.555,A -85,B 0,C 180,E1 -19258.269,E2 -19258.269} C_VEL
LIN {X 0,Y 330.493,Z 894.274,A -85,B 0,C 180,E1 -19261.387,E2 -19261.387} C_VEL
LIN {X 0,Y 330.32,Z 888.236,A -85,B 0,C 180,E1 -19264.514,E2 -19264.514} C_VEL
LIN {X 0,Y 330.554,Z 880.375,A -85,B 0,C 180,E1 -19267.649,E2 -19267.649} C_VEL
LIN {X 0,Y 331.211,Z 870.397,A -85,B 0,C 180,E1 -19270.788,E2 -19270.788} C_VEL
LIN {X 0,Y 332.307,Z 858.864,A -85,B 0,C 180,E1 -19273.751,E2 -19273.751} C_VEL
LIN {X 0,Y 333.832,Z 845.677,A -85,B 0,C 180,E1 -19276.572,E2 -19276.572} C_VEL
LIN {X 0,Y 335.666,Z 831.482,A -85,B 0,C 180,E1 -19279.128,E2 -19279.128} C_VEL
LIN {X 0,Y 337.998,Z 814.487,A -85,B 0,C 180,E1 -19281.702,E2 -19281.702} C_VEL
LIN {X 0,Y 340.647,Z 795.749,A -85,B 0,C 180,E1 -19284.08,E2 -19284.08} C_VEL
LIN {X 0,Y 343.389,Z 775.87,A -85,B 0,C 180,E1 -19286.177,E2 -19286.177} C_VEL
LIN {X 0,Y 346.177,Z 755.006,A -85,B 0,C 180,E1 -19287.993,E2 -19287.993} C_VEL
LIN {X 0,Y 349.023,Z 732.045,A -85,B 0,C 180,E1 -19289.616,E2 -19289.616} C_VEL
LIN {X 0,Y 351.626,Z 708.502,A -85,B 0,C 180,E1 -19290.93,E2 -19290.93} C_VEL
LIN {X 0,Y 353.892,Z 684.83,A -85,B 0,C 180,E1 -19291.924,E2 -19291.924} C_VEL
LIN {X 0,Y 363.226,Z 566.065,A -85,B 0,C 180,E1 -19295.51,E2 -19295.51} C_VEL
LIN {X 0,Y 364.398,Z 565.695,A -85,B 0,C 180,E1 -19295.765,E2 -19295.765} C_VEL
LIN {X 0,Y 366.736,Z 562.036,A -85,B 0,C 180,E1 -19296.117,E2 -19296.117} C_VEL
LIN {X 0,Y 370.609,Z 552.646,A -85,B 0,C 180,E1 -19296.53,E2 -19296.53} C_VEL
LIN {X 0,Y 375.797,Z 536.079,A -85,B 0,C 180,E1 -19296.911,E2 -19296.911} C_VEL
LIN {X 0,Y 376.934,Z 532.398,A -85,B 0,C 180,E1 -19297.001,E2 -19297.001} C_VEL
LIN {X 0,Y 379.856,Z 527.791,A -85,B 0,C 180,E1 -19297.426,E2 -19297.426} C_VEL
LIN {X 0,Y 385.485,Z 514.31,A -85,B 0,C 180,E1 -19298.04,E2 -19298.04} C_VEL
LIN {X 0,Y 387.528,Z 508.554,A -85,B 0,C 180,E1 -19298.238,E2 -19298.238} C_VEL
LIN {X 0,Y 391.2,Z 502.869,A -85,B 0,C 180,E1 -19298.748,E2 -19298.748} C_VEL
LIN {X 0,Y 395.047,Z 494.148,A -85,B 0,C 180,E1 -19299.173,E2 -19299.173} C_VEL
LIN {X 0,Y 397.385,Z 487.686,A -85,B 0,C 180,E1 -19299.398,E2 -19299.398} C_VEL
LIN {X 0,Y 401.539,Z 480.63,A -85,B 0,C 180,E1 -19299.929,E2 -19299.929} C_VEL
LIN {X 0,Y 405.657,Z 470.714,A -85,B 0,C 180,E1 -19300.353,E2 -19300.353} C_VEL
LIN {X 0,Y 406.476,Z 468.475,A -85,B 0,C 180,E1 -19300.431,E2 -19300.431} C_VEL
LIN {X 0,Y 402.319,Z 524.845,A -85,B 0,C 180,E1 -19301.522,E2 -19301.522} C_VEL
LIN {X 0,Y 396.817,Z 580.477,A -85,B 0,C 180,E1 -19302.813,E2 -19302.813} C_VEL
LIN {X 0,Y 390.225,Z 636.395,A -85,B 0,C 180,E1 -19304.359,E2 -19304.359} C_VEL
LIN {X 0,Y 385.459,Z 679.331,A -85,B 0,C 180,E1 -19305.853,E2 -19305.853} C_VEL
LIN {X 0,Y 382.827,Z 700.965,A -85,B 0,C 180,E1 -19306.819,E2 -19306.819} C_VEL
LIN {X 0,Y 379.315,Z 722.606,A -85,B 0,C 180,E1 -19308.069,E2 -19308.069} C_VEL
LIN {X 0,Y 375.208,Z 742.953,A -85,B 0,C 180,E1 -19309.541,E2 -19309.541} C_VEL
LIN {X 0,Y 370.621,Z 762.224,A -85,B 0,C 180,E1 -19311.251,E2 -19311.251} C_VEL
LIN {X 0,Y 365.496,Z 781.044,A -85,B 0,C 180,E1 -19313.28,E2 -19313.28} C_VEL
LIN {X 0,Y 360.132,Z 798.788,A -85,B 0,C 180,E1 -19315.597,E2 -19315.597} C_VEL
LIN {X 0,Y 355.054,Z 814.339,A -85,B 0,C 180,E1 -19318.032,E2 -19318.032} C_VEL
LIN {X 0,Y 349.757,Z 829.623,A -85,B 0,C 180,E1 -19320.922,E2 -19320.922} C_VEL
LIN {X 0,Y 345.024,Z 842.835,A -85,B 0,C 180,E1 -19323.948,E2 -19323.948} C_VEL
LIN {X 0,Y 340.799,Z 854.532,A -85,B 0,C 180,E1 -19327.214,E2 -19327.214} C_VEL
LIN {X 0,Y 337.298,Z 864.397,A -85,B 0,C 180,E1 -19330.609,E2 -19330.609} C_VEL
LIN {X 0,Y 334.407,Z 872.934,A -85,B 0,C 180,E1 -19334.323,E2 -19334.323} C_VEL
LIN {X 0,Y 332.397,Z 879.384,A -85,B 0,C 180,E1 -19338.02,E2 -19338.02} C_VEL
LIN {X 0,Y 331.13,Z 883.931,A -85,B 0,C 180,E1 -19341.666,E2 -19341.666} C_VEL
LIN {X 0,Y 330.454,Z 886.711,A -85,B 0,C 180,E1 -19345.14,E2 -19345.14} C_VEL
LIN {X 0,Y 330.158,Z 888.078,A -85,B 0,C 180,E1 -19348.785,E2 -19348.785} C_VEL
LIN {X 0,Y 330.21,Z 887.92,A -85,B 0,C 180,E1 -19352.256,E2 -19352.256} C_VEL
LIN {X 0,Y 330.607,Z 886.15,A -85,B 0,C 180,E1 -19355.902,E2 -19355.902} C_VEL
LIN {X 0,Y 331.45,Z 882.726,A -85,B 0,C 180,E1 -19359.551,E2 -19359.551} C_VEL
LIN {X 0,Y 332.921,Z 877.621,A -85,B 0,C 180,E1 -19363.194,E2 -19363.194} C_VEL
LIN {X 0,Y 335.132,Z 870.725,A -85,B 0,C 180,E1 -19366.822,E2 -19366.822} C_VEL
LIN {X 0,Y 337.099,Z 865.021,A -85,B 0,C 180,E1 -19369.257,E2 -19369.257} C_VEL
LIN {X 0,Y 337.28,Z 862.137,A -85,B 0,C 180,E1 -19370.481,E2 -19370.481} C_VEL
LIN {X 0,Y 334.683,Z 854.109,A -85,B 0,C 180,E1 -19373.805,E2 -19373.805} C_VEL
LIN {X 0,Y 335.215,Z 850.992,A -85,B 0,C 180,E1 -19374.812,E2 -19374.812} C_VEL
LIN {X 0,Y 339.668,Z 839.224,A -85,B 0,C 180,E1 -19377.908,E2 -19377.908} C_VEL
LIN {X 0,Y 344.597,Z 825.915,A -85,B 0,C 180,E1 -19380.808,E2 -19380.808} C_VEL
LIN {X 0,Y 349.831,Z 811.181,A -85,B 0,C 180,E1 -19383.479,E2 -19383.479} C_VEL
LIN {X 0,Y 355.241,Z 794.915,A -85,B 0,C 180,E1 -19385.934,E2 -19385.934} C_VEL
LIN {X 0,Y 360.526,Z 777.635,A -85,B 0,C 180,E1 -19388.104,E2 -19388.104} C_VEL
LIN {X 0,Y 365.555,Z 759.306,A -85,B 0,C 180,E1 -19390.015,E2 -19390.015} C_VEL
LIN {X 0,Y 370.087,Z 740.299,A -85,B 0,C 180,E1 -19391.654,E2 -19391.654} C_VEL
LIN {X 0,Y 373.931,Z 721.419,A -85,B 0,C 180,E1 -19392.99,E2 -19392.99} C_VEL
LIN {X 0,Y 377.231,Z 701.418,A -85,B 0,C 180,E1 -19394.137,E2 -19394.137} C_VEL
LIN {X 0,Y 379.945,Z 679.696,A -85,B 0,C 180,E1 -19395.108,E2 -19395.108} C_VEL
LIN {X 0,Y 384.883,Z 636.923,A -85,B 0,C 180,E1 -19396.609,E2 -19396.609} C_VEL
LIN {X 0,Y 391.604,Z 581.818,A -85,B 0,C 180,E1 -19398.146,E2 -19398.146} C_VEL
LIN {X 0,Y 397.135,Z 527.059,A -85,B 0,C 180,E1 -19399.42,E2 -19399.42} C_VEL
LIN {X 0,Y 401.186,Z 474.554,A -85,B 0,C 180,E1 -19400.45,E2 -19400.45} C_VEL
LIN {X 0,Y 404.446,Z 425.834,A -85,B 0,C 180,E1 -19401.316,E2 -19401.316} C_VEL
LIN {X 0,Y 411.795,Z 393.606,A -85,B 0,C 180,E1 -19402.449,E2 -19402.449} C_VEL
LIN {X 0,Y 406.174,Z 376.822,A -85,B 0,C 180,E1 -19405.171,E2 -19405.171} C_VEL
LIN {X 0,Y 400.038,Z 360.802,A -85,B 0,C 180,E1 -19408.17,E2 -19408.17} C_VEL
LIN {X 0,Y 394.105,Z 346.94,A -85,B 0,C 180,E1 -19411.18,E2 -19411.18} C_VEL
LIN {X 0,Y 388.507,Z 335.003,A -85,B 0,C 180,E1 -19414.218,E2 -19414.218} C_VEL
LIN {X 0,Y 383.362,Z 325.292,A -85,B 0,C 180,E1 -19417.09,E2 -19417.09} C_VEL
LIN {X 0,Y 378.832,Z 317.185,A -85,B 0,C 180,E1 -19419.852,E2 -19419.852} C_VEL
LIN {X 0,Y 376.064,Z 312.469,A -85,B 0,C 180,E1 -19421.715,E2 -19421.715} C_VEL
LIN {X 0,Y 373.303,Z 307.665,A -85,B 0,C 180,E1 -19423.825,E2 -19423.825} C_VEL
LIN {X 0,Y 370.356,Z 302.809,A -85,B 0,C 180,E1 -19426.256,E2 -19426.256} C_VEL
LIN {X 0,Y 367.881,Z 298.791,A -85,B 0,C 180,E1 -19428.794,E2 -19428.794} C_VEL
LIN {X 0,Y 367.263,Z 297.512,A -85,B 0,C 180,E1 -19429.49,E2 -19429.49} C_VEL
LIN {X 0,Y 364.554,Z 294.322,A -85,B 0,C 180,E1 -19432.593,E2 -19432.593} C_VEL
LIN {X 0,Y 363.716,Z 291.804,A -85,B 0,C 180,E1 -19434.32,E2 -19434.32} C_VEL
LIN {X 0,Y 361.663,Z 289.804,A -85,B 0,C 180,E1 -19441.426,E2 -19441.426} C_VEL
LIN {X 0,Y 362.753,Z 290.696,A -85,B 0,C 180,E1 -19446.171,E2 -19446.171} C_VEL
LIN {X 0,Y 364.756,Z 292.106,A -85,B 0,C 180,E1 -19449.387,E2 -19449.387} C_VEL
LIN {X 0,Y 365.624,Z 297.788,A -85,B 0,C 180,E1 -19451.516,E2 -19451.516} C_VEL
LIN {X 0,Y 367.843,Z 307.216,A -85,B 0,C 180,E1 -19454.683,E2 -19454.683} C_VEL
LIN {X 0,Y 372.203,Z 321.229,A -85,B 0,C 180,E1 -19458.766,E2 -19458.766} C_VEL
LIN {X 0,Y 379.349,Z 340.558,A -85,B 0,C 180,E1 -19463.495,E2 -19463.495} C_VEL
LIN {X 0,Y 385.038,Z 354.114,A -85,B 0,C 180,E1 -19466.343,E2 -19466.343} C_VEL
LIN {X 0,Y 390.121,Z 367.099,A -85,B 0,C 180,E1 -19468.555,E2 -19468.555} C_VEL
LIN {X 0,Y 404.754,Z 390.58,A -85,B 0,C 180,E1 -19471.268,E2 -19471.268} C_VEL
LIN {X 0,Y 382.202,Z 647.493,A -85,B 0,C 180,E1 -19477.208,E2 -19477.208} C_VEL
LIN {X 0,Y 378.254,Z 694.409,A -85,B 0,C 180,E1 -19478.385,E2 -19478.385} C_VEL
LIN {X 0,Y 375.199,Z 718.281,A -85,B 0,C 180,E1 -19479.204,E2 -19479.204} C_VEL
LIN {X 0,Y 371.43,Z 742.34,A -85,B 0,C 180,E1 -19480.279,E2 -19480.279} C_VEL
LIN {X 0,Y 367.2,Z 765.576,A -85,B 0,C 180,E1 -19481.576,E2 -19481.576} C_VEL
LIN {X 0,Y 362.344,Z 788.699,A -85,B 0,C 180,E1 -19483.185,E2 -19483.185} C_VEL
LIN {X 0,Y 357.035,Z 811.648,A -85,B 0,C 180,E1 -19485.116,E2 -19485.116} C_VEL
LIN {X 0,Y 351.826,Z 832.542,A -85,B 0,C 180,E1 -19487.216,E2 -19487.216} C_VEL
LIN {X 0,Y 344.9,Z 860.914,A -85,B 0,C 180,E1 -19490.458,E2 -19490.458} C_VEL
LIN {X 0,Y 340.515,Z 878.143,A -85,B 0,C 180,E1 -19492.835,E2 -19492.835} C_VEL
LIN {X 0,Y 336.3,Z 893.898,A -85,B 0,C 180,E1 -19495.445,E2 -19495.445} C_VEL
LIN {X 0,Y 332.196,Z 908.772,A -85,B 0,C 180,E1 -19498.417,E2 -19498.417} C_VEL
LIN {X 0,Y 328.571,Z 922.264,A -85,B 0,C 180,E1 -19501.658,E2 -19501.658} C_VEL
LIN {X 0,Y 325.611,Z 934.225,A -85,B 0,C 180,E1 -19505.121,E2 -19505.121} C_VEL
LIN {X 0,Y 323.409,Z 944.532,A -85,B 0,C 180,E1 -19508.794,E2 -19508.794} C_VEL
LIN {X 0,Y 322.001,Z 953.295,A -85,B 0,C 180,E1 -19512.656,E2 -19512.656} C_VEL
LIN {X 0,Y 321.334,Z 961.857,A -85,B 0,C 180,E1 -19517.419,E2 -19517.419} C_VEL
LIN {X 0,Y 321.31,Z 967.333,A -85,B 0,C 180,E1 -19521.229,E2 -19521.229} C_VEL
LIN {X 0,Y 321.501,Z 970.682,A -85,B 0,C 180,E1 -19524.468,E2 -19524.468} C_VEL
LIN {X 0,Y 321.63,Z 972.821,A -85,B 0,C 180,E1 -19527.684,E2 -19527.684} C_VEL
LIN {X 0,Y 321.586,Z 973.802,A -85,B 0,C 180,E1 -19531.247,E2 -19531.247} C_VEL
LIN {X 0,Y 321.29,Z 973.303,A -85,B 0,C 180,E1 -19534.641,E2 -19534.641} C_VEL
LIN {X 0,Y 320.963,Z 971.595,A -85,B 0,C 180,E1 -19538.059,E2 -19538.059} C_VEL
LIN {X 0,Y 320.822,Z 968.386,A -85,B 0,C 180,E1 -19541.871,E2 -19541.871} C_VEL
LIN {X 0,Y 321.357,Z 962.923,A -85,B 0,C 180,E1 -19546.262,E2 -19546.262} C_VEL
LIN {X 0,Y 322.761,Z 956.408,A -85,B 0,C 180,E1 -19550.302,E2 -19550.302} C_VEL
LIN {X 0,Y 325.715,Z 947.137,A -85,B 0,C 180,E1 -19554.871,E2 -19554.871} C_VEL
LIN {X 0,Y 330.29,Z 936.141,A -85,B 0,C 180,E1 -19559.323,E2 -19559.323} C_VEL
LIN {X 0,Y 336.456,Z 923.364,A -85,B 0,C 180,E1 -19563.557,E2 -19563.557} C_VEL
LIN {X 0,Y 345.049,Z 907.611,A -85,B 0,C 180,E1 -19567.904,E2 -19567.904} C_VEL
LIN {X 0,Y 354.861,Z 891.066,A -85,B 0,C 180,E1 -19571.695,E2 -19571.695} C_VEL
LIN {X 0,Y 366.402,Z 872.536,A -85,B 0,C 180,E1 -19575.197,E2 -19575.197} C_VEL
LIN {X 0,Y 379.135,Z 852.734,A -85,B 0,C 180,E1 -19578.276,E2 -19578.276} C_VEL
LIN {X 0,Y 393.5,Z 830.922,A -85,B 0,C 180,E1 -19581.037,E2 -19581.037} C_VEL
LIN {X 0,Y 402.533,Z 817.272,A -85,B 0,C 180,E1 -19582.489,E2 -19582.489} C_VEL
LIN {X 0,Y 388.816,Z 833.433,A -85,B 0,C 180,E1 -19584.647,E2 -19584.647} C_VEL
LIN {X 0,Y 375.59,Z 849.152,A -85,B 0,C 180,E1 -19587.287,E2 -19587.287} C_VEL
LIN {X 0,Y 364.132,Z 863.085,A -85,B 0,C 180,E1 -19590.197,E2 -19590.197} C_VEL
LIN {X 0,Y 354.32,Z 875.14,A -85,B 0,C 180,E1 -19593.34,E2 -19593.34} C_VEL
LIN {X 0,Y 346.379,Z 884.782,A -85,B 0,C 180,E1 -19596.524,E2 -19596.524} C_VEL
LIN {X 0,Y 339.731,Z 892.49,A -85,B 0,C 180,E1 -19599.858,E2 -19599.858} C_VEL
LIN {X 0,Y 334.529,Z 897.963,A -85,B 0,C 180,E1 -19603.146,E2 -19603.146} C_VEL
LIN {X 0,Y 330.569,Z 901.446,A -85,B 0,C 180,E1 -19606.353,E2 -19606.353} C_VEL
LIN {X 0,Y 327.503,Z 903.2,A -85,B 0,C 180,E1 -19609.623,E2 -19609.623} C_VEL
LIN {X 0,Y 325.153,Z 903.121,A -85,B 0,C 180,E1 -19613.112,E2 -19613.112} C_VEL
LIN {X 0,Y 323.645,Z 901.16,A -85,B 0,C 180,E1 -19616.457,E2 -19616.457} C_VEL
LIN {X 0,Y 322.794,Z 897.601,A -85,B 0,C 180,E1 -19619.645,E2 -19619.645} C_VEL
LIN {X 0,Y 322.388,Z 892.347,A -85,B 0,C 180,E1 -19622.844,E2 -19622.844} C_VEL
LIN {X 0,Y 322.4,Z 885.246,A -85,B 0,C 180,E1 -19626.053,E2 -19626.053} C_VEL
LIN {X 0,Y 322.842,Z 876.242,A -85,B 0,C 180,E1 -19629.268,E2 -19629.268} C_VEL
LIN {X 0,Y 323.708,Z 865.731,A -85,B 0,C 180,E1 -19632.306,E2 -19632.306} C_VEL
LIN {X 0,Y 325.083,Z 853,A -85,B 0,C 180,E1 -19635.338,E2 -19635.338} C_VEL
LIN {X 0,Y 326.885,Z 838.717,A -85,B 0,C 180,E1 -19638.18,E2 -19638.18} C_VEL
LIN {X 0,Y 329.147,Z 822.349,A -85,B 0,C 180,E1 -19640.913,E2 -19640.913} C_VEL
LIN {X 0,Y 331.661,Z 804.898,A -85,B 0,C 180,E1 -19643.356,E2 -19643.356} C_VEL
LIN {X 0,Y 334.416,Z 785.713,A -85,B 0,C 180,E1 -19645.598,E2 -19645.598} C_VEL
LIN {X 0,Y 337.334,Z 764.634,A -85,B 0,C 180,E1 -19647.638,E2 -19647.638} C_VEL
LIN {X 0,Y 340.268,Z 742.481,A -85,B 0,C 180,E1 -19649.389,E2 -19649.389} C_VEL
LIN {X 0,Y 343.05,Z 719.236,A -85,B 0,C 180,E1 -19650.863,E2 -19650.863} C_VEL
LIN {X 0,Y 345.561,Z 695.392,A -85,B 0,C 180,E1 -19652.03,E2 -19652.03} C_VEL
LIN {X 0,Y 347.887,Z 668.16,A -85,B 0,C 180,E1 -19652.995,E2 -19652.995} C_VEL
LIN {X 0,Y 353.235,Z 601.06,A -85,B 0,C 180,E1 -19655.074,E2 -19655.074} C_VEL
LIN {X 0,Y 354.377,Z 600.785,A -85,B 0,C 180,E1 -19655.339,E2 -19655.339} C_VEL
LIN {X 0,Y 356.658,Z 597.525,A -85,B 0,C 180,E1 -19655.696,E2 -19655.696} C_VEL
LIN {X 0,Y 360.359,Z 589.269,A -85,B 0,C 180,E1 -19656.094,E2 -19656.094} C_VEL
LIN {X 0,Y 365.374,Z 574.567,A -85,B 0,C 180,E1 -19656.445,E2 -19656.445} C_VEL
LIN {X 0,Y 366.315,Z 571.825,A -85,B 0,C 180,E1 -19656.516,E2 -19656.516} C_VEL
LIN {X 0,Y 369.232,Z 567.614,A -85,B 0,C 180,E1 -19656.955,E2 -19656.955} C_VEL
LIN {X 0,Y 373.102,Z 559.212,A -85,B 0,C 180,E1 -19657.386,E2 -19657.386} C_VEL
LIN {X 0,Y 378.287,Z 544.108,A -85,B 0,C 180,E1 -19657.79,E2 -19657.79} C_VEL
LIN {X 0,Y 380.664,Z 536.478,A -85,B 0,C 180,E1 -19657.95,E2 -19657.95} C_VEL
LIN {X 0,Y 384.336,Z 529.971,A -85,B 0,C 180,E1 -19658.421,E2 -19658.421} C_VEL
LIN {X 0,Y 390.486,Z 514.755,A -85,B 0,C 180,E1 -19659.032,E2 -19659.032} C_VEL
LIN {X 0,Y 391.377,Z 512.758,A -85,B 0,C 180,E1 -19659.127,E2 -19659.127} C_VEL
LIN {X 0,Y 395.569,Z 505.766,A -85,B 0,C 180,E1 -19659.662,E2 -19659.662} C_VEL
LIN {X 0,Y 399.483,Z 496.795,A -85,B 0,C 180,E1 -19660.069,E2 -19660.069} C_VEL
LIN {X 0,Y 394.883,Z 549.537,A -85,B 0,C 180,E1 -19661.182,E2 -19661.182} C_VEL
LIN {X 0,Y 388.84,Z 604.249,A -85,B 0,C 180,E1 -19662.554,E2 -19662.554} C_VEL
LIN {X 0,Y 383.007,Z 651.573,A -85,B 0,C 180,E1 -19663.976,E2 -19663.976} C_VEL
LIN {X 0,Y 378.619,Z 690.17,A -85,B 0,C 180,E1 -19665.44,E2 -19665.44} C_VEL
LIN {X 0,Y 375.677,Z 710.691,A -85,B 0,C 180,E1 -19666.474,E2 -19666.474} C_VEL
LIN {X 0,Y 371.933,Z 731.108,A -85,B 0,C 180,E1 -19667.771,E2 -19667.771} C_VEL
LIN {X 0,Y 367.522,Z 751.012,A -85,B 0,C 180,E1 -19669.338,E2 -19669.338} C_VEL
LIN {X 0,Y 362.643,Z 769.877,A -85,B 0,C 180,E1 -19671.151,E2 -19671.151} C_VEL
LIN {X 0,Y 357.426,Z 787.746,A -85,B 0,C 180,E1 -19673.226,E2 -19673.226} C_VEL
LIN {X 0,Y 352.005,Z 804.576,A -85,B 0,C 180,E1 -19675.579,E2 -19675.579} C_VEL
LIN {X 0,Y 346.71,Z 819.846,A -85,B 0,C 180,E1 -19678.146,E2 -19678.146} C_VEL
LIN {X 0,Y 341.668,Z 833.676,A -85,B 0,C 180,E1 -19680.935,E2 -19680.935} C_VEL
LIN {X 0,Y 336.758,Z 846.745,A -85,B 0,C 180,E1 -19684.121,E2 -19684.121} C_VEL
LIN {X 0,Y 332.441,Z 858.175,A -85,B 0,C 180,E1 -19687.543,E2 -19687.543} C_VEL
LIN {X 0,Y 328.822,Z 867.957,A -85,B 0,C 180,E1 -19691.196,E2 -19691.196} C_VEL
LIN {X 0,Y 326.036,Z 875.95,A -85,B 0,C 180,E1 -19695.027,E2 -19695.027} C_VEL
LIN {X 0,Y 324.137,Z 881.846,A -85,B 0,C 180,E1 -19698.803,E2 -19698.803} C_VEL
LIN {X 0,Y 322.991,Z 885.922,A -85,B 0,C 180,E1 -19702.529,E2 -19702.529} C_VEL
LIN {X 0,Y 322.411,Z 888.316,A -85,B 0,C 180,E1 -19706.088,E2 -19706.088} C_VEL
LIN {X 0,Y 322.213,Z 889.207,A -85,B 0,C 180,E1 -19709.822,E2 -19709.822} C_VEL
LIN {X 0,Y 322.344,Z 888.541,A -85,B 0,C 180,E1 -19713.379,E2 -19713.379} C_VEL
LIN {X 0,Y 322.894,Z 886.307,A -85,B 0,C 180,E1 -19717.115,E2 -19717.115} C_VEL
LIN {X 0,Y 323.974,Z 882.449,A -85,B 0,C 180,E1 -19720.852,E2 -19720.852} C_VEL
LIN {X 0,Y 325.657,Z 877.203,A -85,B 0,C 180,E1 -19724.401,E2 -19724.401} C_VEL
LIN {X 0,Y 328.184,Z 869.891,A -85,B 0,C 180,E1 -19728.105,E2 -19728.105} C_VEL
LIN {X 0,Y 331.613,Z 860.58,A -85,B 0,C 180,E1 -19731.769,E2 -19731.769} C_VEL
LIN {X 0,Y 335.215,Z 850.992,A -85,B 0,C 180,E1 -19734.812,E2 -19734.812} C_VEL
LIN {X 0,Y 335.806,Z 847.302,A -85,B 0,C 180,E1 -19735.975,E2 -19735.975} C_VEL
LIN {X 0,Y 334.369,Z 837.952,A -85,B 0,C 180,E1 -19739.006,E2 -19739.006} C_VEL
LIN {X 0,Y 335.24,Z 833.575,A -85,B 0,C 180,E1 -19740.104,E2 -19740.104} C_VEL
LIN {X 0,Y 340.501,Z 819.67,A -85,B 0,C 180,E1 -19742.906,E2 -19742.906} C_VEL
LIN {X 0,Y 345.707,Z 805.162,A -85,B 0,C 180,E1 -19745.35,E2 -19745.35} C_VEL
LIN {X 0,Y 351.333,Z 788.291,A -85,B 0,C 180,E1 -19747.726,E2 -19747.726} C_VEL
LIN {X 0,Y 356.785,Z 770.221,A -85,B 0,C 180,E1 -19749.835,E2 -19749.835} C_VEL
LIN {X 0,Y 361.814,Z 751.331,A -85,B 0,C 180,E1 -19751.654,E2 -19751.654} C_VEL
LIN {X 0,Y 366.386,Z 731.238,A -85,B 0,C 180,E1 -19753.235,E2 -19753.235} C_VEL
LIN {X 0,Y 370.253,Z 710.53,A -85,B 0,C 180,E1 -19754.545,E2 -19754.545} C_VEL
LIN {X 0,Y 373.355,Z 688.971,A -85,B 0,C 180,E1 -19755.614,E2 -19755.614} C_VEL
LIN {X 0,Y 378.118,Z 648.948,A -85,B 0,C 180,E1 -19757.124,E2 -19757.124} C_VEL
LIN {X 0,Y 384.174,Z 601.052,A -85,B 0,C 180,E1 -19758.547,E2 -19758.547} C_VEL
LIN {X 0,Y 390.361,Z 545.706,A -85,B 0,C 180,E1 -19759.921,E2 -19759.921} C_VEL
LIN {X 0,Y 394.842,Z 494.374,A -85,B 0,C 180,E1 -19760.991,E2 -19760.991} C_VEL
LIN {X 0,Y 399.349,Z 428.731,A -85,B 0,C 180,E1 -19762.169,E2 -19762.169} C_VEL
LIN {X 0,Y 406.606,Z 397.088,A -85,B 0,C 180,E1 -19763.26,E2 -19763.26} C_VEL
LIN {X 0,Y 401.35,Z 381.205,A -85,B 0,C 180,E1 -19765.906,E2 -19765.906} C_VEL
LIN {X 0,Y 395.659,Z 366.11,A -85,B 0,C 180,E1 -19768.797,E2 -19768.797} C_VEL
LIN {X 0,Y 390.132,Z 352.976,A -85,B 0,C 180,E1 -19771.696,E2 -19771.696} C_VEL
LIN {X 0,Y 384.975,Z 341.645,A -85,B 0,C 180,E1 -19774.624,E2 -19774.624} C_VEL
LIN {X 0,Y 380.102,Z 332.089,A -85,B 0,C 180,E1 -19777.496,E2 -19777.496} C_VEL
LIN {X 0,Y 375.733,Z 324.127,A -85,B 0,C 180,E1 -19780.247,E2 -19780.247} C_VEL
LIN {X 0,Y 373.065,Z 319.456,A -85,B 0,C 180,E1 -19782.128,E2 -19782.128} C_VEL
LIN {X 0,Y 370.614,Z 314.988,A -85,B 0,C 180,E1 -19784.107,E2 -19784.107} C_VEL
LIN {X 0,Y 367.877,Z 310.29,A -85,B 0,C 180,E1 -19786.482,E2 -19786.482} C_VEL
LIN {X 0,Y 365.476,Z 306.133,A -85,B 0,C 180,E1 -19789.119,E2 -19789.119} C_VEL
LIN {X 0,Y 364.988,Z 305.086,A -85,B 0,C 180,E1 -19789.743,E2 -19789.743} C_VEL
LIN {X 0,Y 362.386,Z 301.831,A -85,B 0,C 180,E1 -19792.868,E2 -19792.868} C_VEL
LIN {X 0,Y 361.666,Z 299.521,A -85,B 0,C 180,E1 -19794.447,E2 -19794.447} C_VEL
LIN {X 0,Y 359.843,Z 297.595,A -85,B 0,C 180,E1 -19801.433,E2 -19801.433} C_VEL
LIN {X 0,Y 361.042,Z 298.525,A -85,B 0,C 180,E1 -19806.201,E2 -19806.201} C_VEL
LIN {X 0,Y 362.837,Z 299.912,A -85,B 0,C 180,E1 -19809.197,E2 -19809.197} C_VEL
LIN {X 0,Y 364.105,Z 307.723,A -85,B 0,C 180,E1 -19812.047,E2 -19812.047} C_VEL
LIN {X 0,Y 366.044,Z 315.833,A -85,B 0,C 180,E1 -19814.676,E2 -19814.676} C_VEL
LIN {X 0,Y 369.783,Z 328.376,A -85,B 0,C 180,E1 -19818.337,E2 -19818.337} C_VEL
LIN {X 0,Y 376.578,Z 347.233,A -85,B 0,C 180,E1 -19822.974,E2 -19822.974} C_VEL
LIN {X 0,Y 381.903,Z 360.372,A -85,B 0,C 180,E1 -19825.761,E2 -19825.761} C_VEL
LIN {X 0,Y 388.582,Z 377.895,A -85,B 0,C 180,E1 -19828.742,E2 -19828.742} C_VEL
LIN {X 0,Y 398.412,Z 393.907,A -85,B 0,C 180,E1 -19830.591,E2 -19830.591} C_VEL
LIN {X 0,Y 373.667,Z 668.611,A -85,B 0,C 180,E1 -19837.092,E2 -19837.092} C_VEL
LIN {X 0,Y 370.77,Z 698.909,A -85,B 0,C 180,E1 -19837.918,E2 -19837.918} C_VEL
LIN {X 0,Y 367.548,Z 722.861,A -85,B 0,C 180,E1 -19838.788,E2 -19838.788} C_VEL
LIN {X 0,Y 363.541,Z 746.89,A -85,B 0,C 180,E1 -19839.943,E2 -19839.943} C_VEL
LIN {X 0,Y 358.932,Z 770.714,A -85,B 0,C 180,E1 -19841.375,E2 -19841.375} C_VEL
LIN {X 0,Y 354.087,Z 792.961,A -85,B 0,C 180,E1 -19842.998,E2 -19842.998} C_VEL
LIN {X 0,Y 348.844,Z 814.672,A -85,B 0,C 180,E1 -19844.93,E2 -19844.93} C_VEL
LIN {X 0,Y 342.947,Z 841.315,A -85,B 0,C 180,E1 -19847.436,E2 -19847.436} C_VEL
LIN {X 0,Y 338.565,Z 859.044,A -85,B 0,C 180,E1 -19849.479,E2 -19849.479} C_VEL
LIN {X 0,Y 334.073,Z 875.956,A -85,B 0,C 180,E1 -19851.825,E2 -19851.825} C_VEL
LIN {X 0,Y 329.719,Z 891.424,A -85,B 0,C 180,E1 -19854.391,E2 -19854.391} C_VEL
LIN {X 0,Y 325.413,Z 906.23,A -85,B 0,C 180,E1 -19857.343,E2 -19857.343} C_VEL
LIN {X 0,Y 321.568,Z 919.684,A -85,B 0,C 180,E1 -19860.575,E2 -19860.575} C_VEL
LIN {X 0,Y 318.306,Z 931.885,A -85,B 0,C 180,E1 -19864.11,E2 -19864.11} C_VEL
LIN {X 0,Y 315.936,Z 942.016,A -85,B 0,C 180,E1 -19867.68,E2 -19867.68} C_VEL
LIN {X 0,Y 314.285,Z 951.055,A -85,B 0,C 180,E1 -19871.641,E2 -19871.641} C_VEL
LIN {X 0,Y 313.503,Z 958.173,A -85,B 0,C 180,E1 -19875.595,E2 -19875.595} C_VEL
LIN {X 0,Y 313.371,Z 965.46,A -85,B 0,C 180,E1 -19880.635,E2 -19880.635} C_VEL
LIN {X 0,Y 313.578,Z 969.332,A -85,B 0,C 180,E1 -19884.327,E2 -19884.327} C_VEL
LIN {X 0,Y 313.718,Z 971.463,A -85,B 0,C 180,E1 -19887.443,E2 -19887.443} C_VEL
LIN {X 0,Y 313.699,Z 972.514,A -85,B 0,C 180,E1 -19890.548,E2 -19890.548} C_VEL
LIN {X 0,Y 313.427,Z 972.468,A -85,B 0,C 180,E1 -19894.025,E2 -19894.025} C_VEL
LIN {X 0,Y 313.02,Z 970.857,A -85,B 0,C 180,E1 -19897.895,E2 -19897.895} C_VEL
LIN {X 0,Y 312.839,Z 967.991,A -85,B 0,C 180,E1 -19901.617,E2 -19901.617} C_VEL
LIN {X 0,Y 313.249,Z 963.47,A -85,B 0,C 180,E1 -19905.743,E2 -19905.743} C_VEL
LIN {X 0,Y 314.719,Z 956.729,A -85,B 0,C 180,E1 -19910.262,E2 -19910.262} C_VEL
LIN {X 0,Y 317.559,Z 948.375,A -85,B 0,C 180,E1 -19914.757,E2 -19914.757} C_VEL
LIN {X 0,Y 322.2,Z 937.7,A -85,B 0,C 180,E1 -19919.362,E2 -19919.362} C_VEL
LIN {X 0,Y 328.995,Z 924.676,A -85,B 0,C 180,E1 -19924.002,E2 -19924.002} C_VEL
LIN {X 0,Y 337.596,Z 910.093,A -85,B 0,C 180,E1 -19928.29,E2 -19928.29} C_VEL
LIN {X 0,Y 347.982,Z 893.721,A -85,B 0,C 180,E1 -19932.251,E2 -19932.251} C_VEL
LIN {X 0,Y 360.429,Z 875.269,A -85,B 0,C 180,E1 -19935.932,E2 -19935.932} C_VEL
LIN {X 0,Y 373.911,Z 856.085,A -85,B 0,C 180,E1 -19939.068,E2 -19939.068} C_VEL
LIN {X 0,Y 389.053,Z 835.026,A -85,B 0,C 180,E1 -19941.854,E2 -19941.854} C_VEL
LIN {X 0,Y 393.229,Z 829.126,A -85,B 0,C 180,E1 -19942.543,E2 -19942.543} C_VEL
LIN {X 0,Y 378.6,Z 844.84,A -85,B 0,C 180,E1 -19944.957,E2 -19944.957} C_VEL
LIN {X 0,Y 364.829,Z 859.877,A -85,B 0,C 180,E1 -19947.88,E2 -19947.88} C_VEL
LIN {X 0,Y 353.199,Z 872.771,A -85,B 0,C 180,E1 -19951.047,E2 -19951.047} C_VEL
LIN {X 0,Y 343.722,Z 883.267,A -85,B 0,C 180,E1 -19954.314,E2 -19954.314} C_VEL
LIN {X 0,Y 336.086,Z 891.463,A -85,B 0,C 180,E1 -19957.616,E2 -19957.616} C_VEL
LIN {X 0,Y 330.01,Z 897.493,A -85,B 0,C 180,E1 -19960.899,E2 -19960.899} C_VEL
LIN {X 0,Y 325.055,Z 901.743,A -85,B 0,C 180,E1 -19964.294,E2 -19964.294} C_VEL
LIN {X 0,Y 321.344,Z 904.085,A -85,B 0,C 180,E1 -19967.602,E2 -19967.602} C_VEL
LIN {X 0,Y 318.546,Z 904.725,A -85,B 0,C 180,E1 -19970.97,E2 -19970.97} C_VEL
LIN {X 0,Y 316.543,Z 903.592,A -85,B 0,C 180,E1 -19974.38,E2 -19974.38} C_VEL
LIN {X 0,Y 315.25,Z 900.615,A -85,B 0,C 180,E1 -19977.819,E2 -19977.819} C_VEL
LIN {X 0,Y 314.585,Z 896.074,A -85,B 0,C 180,E1 -19981.093,E2 -19981.093} C_VEL
LIN {X 0,Y 314.363,Z 889.809,A -85,B 0,C 180,E1 -19984.378,E2 -19984.378} C_VEL
LIN {X 0,Y 314.561,Z 882.135,A -85,B 0,C 180,E1 -19987.489,E2 -19987.489} C_VEL
LIN {X 0,Y 315.17,Z 872.642,A -85,B 0,C 180,E1 -19990.603,E2 -19990.603} C_VEL
LIN {X 0,Y 316.272,Z 861.168,A -85,B 0,C 180,E1 -19993.716,E2 -19993.716} C_VEL
LIN {X 0,Y 317.81,Z 848.196,A -85,B 0,C 180,E1 -19996.637,E2 -19996.637} C_VEL
LIN {X 0,Y 319.873,Z 832.797,A -85,B 0,C 180,E1 -19999.54,E2 -19999.54} C_VEL
LIN {X 0,Y 322.331,Z 815.748,A -85,B 0,C 180,E1 -20002.238,E2 -20002.238} C_VEL
LIN {X 0,Y 325.123,Z 796.996,A -85,B 0,C 180,E1 -20004.725,E2 -20004.725} C_VEL
LIN {X 0,Y 328.019,Z 777.192,A -85,B 0,C 180,E1 -20006.915,E2 -20006.915} C_VEL
LIN {X 0,Y 330.97,Z 756.171,A -85,B 0,C 180,E1 -20008.822,E2 -20008.822} C_VEL
LIN {X 0,Y 333.937,Z 733.443,A -85,B 0,C 180,E1 -20010.499,E2 -20010.499} C_VEL
LIN {X 0,Y 336.653,Z 710.193,A -85,B 0,C 180,E1 -20011.861,E2 -20011.861} C_VEL
LIN {X 0,Y 339.159,Z 685.708,A -85,B 0,C 180,E1 -20012.952,E2 -20012.952} C_VEL
LIN {X 0,Y 343.478,Z 632.653,A -85,B 0,C 180,E1 -20014.689,E2 -20014.689} C_VEL
LIN {X 0,Y 344.735,Z 632.45,A -85,B 0,C 180,E1 -20015,E2 -20015} C_VEL
LIN {X 0,Y 347.033,Z 629.365,A -85,B 0,C 180,E1 -20015.367,E2 -20015.367} C_VEL
LIN {X 0,Y 350.778,Z 621.496,A -85,B 0,C 180,E1 -20015.77,E2 -20015.77} C_VEL
LIN {X 0,Y 355.643,Z 608.037,A -85,B 0,C 180,E1 -20016.087,E2 -20016.087} C_VEL
LIN {X 0,Y 356.115,Z 606.902,A -85,B 0,C 180,E1 -20016.131,E2 -20016.131} C_VEL
LIN {X 0,Y 359.152,Z 602.741,A -85,B 0,C 180,E1 -20016.594,E2 -20016.594} C_VEL
LIN {X 0,Y 363.027,Z 594.841,A -85,B 0,C 180,E1 -20017.017,E2 -20017.017} C_VEL
LIN {X 0,Y 368.138,Z 580.915,A -85,B 0,C 180,E1 -20017.395,E2 -20017.395} C_VEL
LIN {X 0,Y 369.769,Z 576.111,A -85,B 0,C 180,E1 -20017.5,E2 -20017.5} C_VEL
LIN {X 0,Y 373.573,Z 569.906,A -85,B 0,C 180,E1 -20017.996,E2 -20017.996} C_VEL
LIN {X 0,Y 378.079,Z 559.492,A -85,B 0,C 180,E1 -20018.438,E2 -20018.438} C_VEL
LIN {X 0,Y 383.632,Z 542.779,A -85,B 0,C 180,E1 -20018.812,E2 -20018.812} C_VEL
LIN {X 0,Y 384.603,Z 540.122,A -85,B 0,C 180,E1 -20018.892,E2 -20018.892} C_VEL
LIN {X 0,Y 388.796,Z 532.262,A -85,B 0,C 180,E1 -20019.377,E2 -20019.377} C_VEL
LIN {X 0,Y 392.244,Z 524.301,A -85,B 0,C 180,E1 -20019.718,E2 -20019.718} C_VEL
LIN {X 0,Y 386.565,Z 579.919,A -85,B 0,C 180,E1 -20021.005,E2 -20021.005} C_VEL
LIN {X 0,Y 379.576,Z 636.233,A -85,B 0,C 180,E1 -20022.571,E2 -20022.571} C_VEL
LIN {X 0,Y 374.411,Z 678.98,A -85,B 0,C 180,E1 -20024.079,E2 -20024.079} C_VEL
LIN {X 0,Y 371.527,Z 701.631,A -85,B 0,C 180,E1 -20025.087,E2 -20025.087} C_VEL
LIN {X 0,Y 368.038,Z 722.338,A -85,B 0,C 180,E1 -20026.276,E2 -20026.276} C_VEL
LIN {X 0,Y 363.901,Z 742.055,A -85,B 0,C 180,E1 -20027.686,E2 -20027.686} C_VEL
LIN {X 0,Y 359.056,Z 761.63,A -85,B 0,C 180,E1 -20029.407,E2 -20029.407} C_VEL
LIN {X 0,Y 353.845,Z 779.885,A -85,B 0,C 180,E1 -20031.354,E2 -20031.354} C_VEL
LIN {X 0,Y 348.221,Z 797.552,A -85,B 0,C 180,E1 -20033.633,E2 -20033.633} C_VEL
LIN {X 0,Y 342.656,Z 813.579,A -85,B 0,C 180,E1 -20036.127,E2 -20036.127} C_VEL
LIN {X 0,Y 337.111,Z 828.512,A -85,B 0,C 180,E1 -20038.929,E2 -20038.929} C_VEL
LIN {X 0,Y 331.922,Z 841.898,A -85,B 0,C 180,E1 -20041.97,E2 -20041.97} C_VEL
LIN {X 0,Y 327.221,Z 853.771,A -85,B 0,C 180,E1 -20045.252,E2 -20045.252} C_VEL
LIN {X 0,Y 323.136,Z 864.127,A -85,B 0,C 180,E1 -20048.774,E2 -20048.774} C_VEL
LIN {X 0,Y 319.793,Z 872.911,A -85,B 0,C 180,E1 -20052.533,E2 -20052.533} C_VEL
LIN {X 0,Y 317.351,Z 879.758,A -85,B 0,C 180,E1 -20056.331,E2 -20056.331} C_VEL
LIN {X 0,Y 315.718,Z 884.817,A -85,B 0,C 180,E1 -20060.153,E2 -20060.153} C_VEL
LIN {X 0,Y 314.775,Z 888.2,A -85,B 0,C 180,E1 -20063.983,E2 -20063.983} C_VEL
LIN {X 0,Y 314.338,Z 889.944,A -85,B 0,C 180,E1 -20067.812,E2 -20067.812} C_VEL
LIN {X 0,Y 314.291,Z 890.073,A -85,B 0,C 180,E1 -20071.458,E2 -20071.458} C_VEL
LIN {X 0,Y 314.639,Z 888.678,A -85,B 0,C 180,E1 -20075.288,E2 -20075.288} C_VEL
LIN {X 0,Y 315.461,Z 885.688,A -85,B 0,C 180,E1 -20079.119,E2 -20079.119} C_VEL
LIN {X 0,Y 316.902,Z 881.182,A -85,B 0,C 180,E1 -20082.848,E2 -20082.848} C_VEL
LIN {X 0,Y 319.088,Z 874.987,A -85,B 0,C 180,E1 -20086.568,E2 -20086.568} C_VEL
LIN {X 0,Y 322.201,Z 866.746,A -85,B 0,C 180,E1 -20090.339,E2 -20090.339} C_VEL
LIN {X 0,Y 326.258,Z 856.419,A -85,B 0,C 180,E1 -20094.055,E2 -20094.055} C_VEL
LIN {X 0,Y 330.771,Z 845.057,A -85,B 0,C 180,E1 -20097.354,E2 -20097.354} C_VEL
LIN {X 0,Y 335.24,Z 833.575,A -85,B 0,C 180,E1 -20100.104,E2 -20100.104} C_VEL
LIN {X 0,Y 336.184,Z 829.154,A -85,B 0,C 180,E1 -20101.182,E2 -20101.182} C_VEL
LIN {X 0,Y 335.663,Z 818.053,A -85,B 0,C 180,E1 -20104.035,E2 -20104.035} C_VEL
LIN {X 0,Y 336.78,Z 812.978,A -85,B 0,C 180,E1 -20105.029,E2 -20105.029} C_VEL
LIN {X 0,Y 342.488,Z 797.034,A -85,B 0,C 180,E1 -20107.496,E2 -20107.496} C_VEL
LIN {X 0,Y 348.159,Z 779.744,A -85,B 0,C 180,E1 -20109.718,E2 -20109.718} C_VEL
LIN {X 0,Y 353.502,Z 761.486,A -85,B 0,C 180,E1 -20111.659,E2 -20111.659} C_VEL
LIN {X 0,Y 358.371,Z 742.286,A -85,B 0,C 180,E1 -20113.343,E2 -20113.343} C_VEL
LIN {X 0,Y 362.464,Z 723.279,A -85,B 0,C 180,E1 -20114.704,E2 -20114.704} C_VEL
LIN {X 0,Y 365.923,Z 703.4,A -85,B 0,C 180,E1 -20115.856,E2 -20115.856} C_VEL
LIN {X 0,Y 368.769,Z 681.99,A -85,B 0,C 180,E1 -20116.827,E2 -20116.827} C_VEL
LIN {X 0,Y 374.11,Z 639.161,A -85,B 0,C 180,E1 -20118.372,E2 -20118.372} C_VEL
LIN {X 0,Y 380.911,Z 586.596,A -85,B 0,C 180,E1 -20119.865,E2 -20119.865} C_VEL
LIN {X 0,Y 386.649,Z 533.162,A -85,B 0,C 180,E1 -20121.129,E2 -20121.129} C_VEL
LIN {X 0,Y 390.902,Z 481.335,A -85,B 0,C 180,E1 -20122.159,E2 -20122.159} C_VEL
LIN {X 0,Y 394.417,Z 431.388,A -85,B 0,C 180,E1 -20123.053,E2 -20123.053} C_VEL
LIN {X 0,Y 401.497,Z 400.6,A -85,B 0,C 180,E1 -20124.096,E2 -20124.096} C_VEL
LIN {X 0,Y 396.31,Z 384.825,A -85,B 0,C 180,E1 -20126.805,E2 -20126.805} C_VEL
LIN {X 0,Y 390.804,Z 370.04,A -85,B 0,C 180,E1 -20129.733,E2 -20129.733} C_VEL
LIN {X 0,Y 385.213,Z 356.616,A -85,B 0,C 180,E1 -20132.816,E2 -20132.816} C_VEL
LIN {X 0,Y 379.626,Z 344.486,A -85,B 0,C 180,E1 -20136.111,E2 -20136.111} C_VEL
LIN {X 0,Y 374.863,Z 335.107,A -85,B 0,C 180,E1 -20139.18,E2 -20139.18} C_VEL
LIN {X 0,Y 370.904,Z 327.545,A -85,B 0,C 180,E1 -20142.021,E2 -20142.021} C_VEL
LIN {X 0,Y 367.713,Z 322.04,A -85,B 0,C 180,E1 -20144.545,E2 -20144.545} C_VEL
LIN {X 0,Y 365.231,Z 317.579,A -85,B 0,C 180,E1 -20146.866,E2 -20146.866} C_VEL
LIN {X 0,Y 362.946,Z 313.195,A -85,B 0,C 180,E1 -20149.58,E2 -20149.58} C_VEL
LIN {X 0,Y 360.105,Z 309.008,A -85,B 0,C 180,E1 -20153.383,E2 -20153.383} C_VEL
LIN {X 0,Y 359.553,Z 307.196,A -85,B 0,C 180,E1 -20154.734,E2 -20154.734} C_VEL
LIN {X 0,Y 358.044,Z 305.424,A -85,B 0,C 180,E1 -20161.12,E2 -20161.12} C_VEL
LIN {X 0,Y 359,Z 306.071,A -85,B 0,C 180,E1 -20165.434,E2 -20165.434} C_VEL
LIN {X 0,Y 361.012,Z 307.722,A -85,B 0,C 180,E1 -20169.003,E2 -20169.003} C_VEL
LIN {X 0,Y 363.253,Z 320.836,A -85,B 0,C 180,E1 -20173.572,E2 -20173.572} C_VEL
LIN {X 0,Y 367.234,Z 334.978,A -85,B 0,C 180,E1 -20177.755,E2 -20177.755} C_VEL
LIN {X 0,Y 374.146,Z 354.706,A -85,B 0,C 180,E1 -20182.634,E2 -20182.634} C_VEL
LIN {X 0,Y 378.877,Z 366.831,A -85,B 0,C 180,E1 -20185.207,E2 -20185.207} C_VEL
LIN {X 0,Y 387.037,Z 388.694,A -85,B 0,C 180,E1 -20188.931,E2 -20188.931} C_VEL
LIN {X 0,Y 392.039,Z 397.2,A -85,B 0,C 180,E1 -20189.906,E2 -20189.906} C_VEL
LIN {X 0,Y 364.652,Z 692.358,A -85,B 0,C 180,E1 -20197.081,E2 -20197.081} C_VEL
LIN {X 0,Y 361.368,Z 717.115,A -85,B 0,C 180,E1 -20197.953,E2 -20197.953} C_VEL
LIN {X 0,Y 357.136,Z 742.873,A -85,B 0,C 180,E1 -20199.147,E2 -20199.147} C_VEL
LIN {X 0,Y 352.587,Z 766.526,A -85,B 0,C 180,E1 -20200.535,E2 -20200.535} C_VEL
LIN {X 0,Y 347.545,Z 789.471,A -85,B 0,C 180,E1 -20202.198,E2 -20202.198} C_VEL
LIN {X 0,Y 344.555,Z 803.046,A -85,B 0,C 180,E1 -20203.248,E2 -20203.248} C_VEL
LIN {X 0,Y 340.408,Z 824.125,A -85,B 0,C 180,E1 -20204.936,E2 -20204.936} C_VEL
LIN {X 0,Y 336.038,Z 843.172,A -85,B 0,C 180,E1 -20206.814,E2 -20206.814} C_VEL
LIN {X 0,Y 331.289,Z 861.282,A -85,B 0,C 180,E1 -20208.986,E2 -20208.986} C_VEL
LIN {X 0,Y 326.455,Z 878.195,A -85,B 0,C 180,E1 -20211.463,E2 -20211.463} C_VEL
LIN {X 0,Y 321.707,Z 893.976,A -85,B 0,C 180,E1 -20214.245,E2 -20214.245} C_VEL
LIN {X 0,Y 317.312,Z 908.347,A -85,B 0,C 180,E1 -20217.284,E2 -20217.284} C_VEL
LIN {X 0,Y 313.439,Z 921.294,A -85,B 0,C 180,E1 -20220.576,E2 -20220.576} C_VEL
LIN {X 0,Y 310.158,Z 933.006,A -85,B 0,C 180,E1 -20224.201,E2 -20224.201} C_VEL
LIN {X 0,Y 307.705,Z 943.212,A -85,B 0,C 180,E1 -20228.056,E2 -20228.056} C_VEL
LIN {X 0,Y 306.136,Z 951.866,A -85,B 0,C 180,E1 -20232.12,E2 -20232.12} C_VEL
LIN {X 0,Y 305.459,Z 958.533,A -85,B 0,C 180,E1 -20236.175,E2 -20236.175} C_VEL
LIN {X 0,Y 305.478,Z 964.84,A -85,B 0,C 180,E1 -20241.151,E2 -20241.151} C_VEL
LIN {X 0,Y 305.703,Z 968.418,A -85,B 0,C 180,E1 -20244.745,E2 -20244.745} C_VEL
LIN {X 0,Y 305.829,Z 970.462,A -85,B 0,C 180,E1 -20247.939,E2 -20247.939} C_VEL
LIN {X 0,Y 305.756,Z 971.45,A -85,B 0,C 180,E1 -20251.312,E2 -20251.312} C_VEL
LIN {X 0,Y 305.373,Z 971.154,A -85,B 0,C 180,E1 -20255.072,E2 -20255.072} C_VEL
LIN {X 0,Y 304.984,Z 969.394,A -85,B 0,C 180,E1 -20258.864,E2 -20258.864} C_VEL
LIN {X 0,Y 304.909,Z 966.391,A -85,B 0,C 180,E1 -20262.692,E2 -20262.692} C_VEL
LIN {X 0,Y 305.667,Z 960.934,A -85,B 0,C 180,E1 -20267.515,E2 -20267.515} C_VEL
LIN {X 0,Y 307.568,Z 954.22,A -85,B 0,C 180,E1 -20271.954,E2 -20271.954} C_VEL
LIN {X 0,Y 311.587,Z 944.396,A -85,B 0,C 180,E1 -20277.109,E2 -20277.109} C_VEL
LIN {X 0,Y 317.503,Z 933.001,A -85,B 0,C 180,E1 -20281.943,E2 -20281.943} C_VEL
LIN {X 0,Y 325.535,Z 919.507,A -85,B 0,C 180,E1 -20286.575,E2 -20286.575} C_VEL
LIN {X 0,Y 335.726,Z 904.12,A -85,B 0,C 180,E1 -20290.937,E2 -20290.937} C_VEL
LIN {X 0,Y 347.595,Z 887.511,A -85,B 0,C 180,E1 -20294.811,E2 -20294.811} C_VEL
LIN {X 0,Y 361.409,Z 869.003,A -85,B 0,C 180,E1 -20298.331,E2 -20298.331} C_VEL
LIN {X 0,Y 376.495,Z 849.461,A -85,B 0,C 180,E1 -20301.334,E2 -20301.334} C_VEL
LIN {X 0,Y 383.915,Z 840.004,A -85,B 0,C 180,E1 -20302.592,E2 -20302.592} C_VEL
LIN {X 0,Y 369.097,Z 854.575,A -85,B 0,C 180,E1 -20305.138,E2 -20305.138} C_VEL
LIN {X 0,Y 355.676,Z 867.956,A -85,B 0,C 180,E1 -20308.095,E2 -20308.095} C_VEL
LIN {X 0,Y 343.648,Z 880.049,A -85,B 0,C 180,E1 -20311.498,E2 -20311.498} C_VEL
LIN {X 0,Y 334.295,Z 889.299,A -85,B 0,C 180,E1 -20314.866,E2 -20314.866} C_VEL
LIN {X 0,Y 326.776,Z 896.357,A -85,B 0,C 180,E1 -20318.269,E2 -20318.269} C_VEL
LIN {X 0,Y 320.566,Z 901.556,A -85,B 0,C 180,E1 -20321.825,E2 -20321.825} C_VEL
LIN {X 0,Y 315.822,Z 904.707,A -85,B 0,C 180,E1 -20325.328,E2 -20325.328} C_VEL
LIN {X 0,Y 312.335,Z 906.022,A -85,B 0,C 180,E1 -20328.739,E2 -20328.739} C_VEL
LIN {X 0,Y 309.765,Z 905.647,A -85,B 0,C 180,E1 -20332.208,E2 -20332.208} C_VEL
LIN {X 0,Y 307.992,Z 903.488,A -85,B 0,C 180,E1 -20335.718,E2 -20335.718} C_VEL
LIN {X 0,Y 306.93,Z 899.49,A -85,B 0,C 180,E1 -20339.253,E2 -20339.253} C_VEL
LIN {X 0,Y 306.445,Z 893.956,A -85,B 0,C 180,E1 -20342.618,E2 -20342.618} C_VEL
LIN {X 0,Y 306.43,Z 886.643,A -85,B 0,C 180,E1 -20345.994,E2 -20345.994} C_VEL
LIN {X 0,Y 306.843,Z 877.905,A -85,B 0,C 180,E1 -20349.188,E2 -20349.188} C_VEL
LIN {X 0,Y 307.726,Z 867.204,A -85,B 0,C 180,E1 -20352.384,E2 -20352.384} C_VEL
LIN {X 0,Y 309.068,Z 855.123,A -85,B 0,C 180,E1 -20355.402,E2 -20355.402} C_VEL
LIN {X 0,Y 310.917,Z 840.993,A -85,B 0,C 180,E1 -20358.371,E2 -20358.371} C_VEL
LIN {X 0,Y 313.265,Z 824.574,A -85,B 0,C 180,E1 -20361.248,E2 -20361.248} C_VEL
LIN {X 0,Y 315.979,Z 806.581,A -85,B 0,C 180,E1 -20363.894,E2 -20363.894} C_VEL
LIN {X 0,Y 318.981,Z 786.801,A -85,B 0,C 180,E1 -20366.321,E2 -20366.321} C_VEL
LIN {X 0,Y 322.073,Z 765.694,A -85,B 0,C 180,E1 -20368.46,E2 -20368.46} C_VEL
LIN {X 0,Y 325.317,Z 742.556,A -85,B 0,C 180,E1 -20370.372,E2 -20370.372} C_VEL
LIN {X 0,Y 328.168,Z 720.019,A -85,B 0,C 180,E1 -20371.862,E2 -20371.862} C_VEL
LIN {X 0,Y 330.862,Z 695.808,A -85,B 0,C 180,E1 -20373.099,E2 -20373.099} C_VEL
LIN {X 0,Y 333.298,Z 668.83,A -85,B 0,C 180,E1 -20374.099,E2 -20374.099} C_VEL
LIN {X 0,Y 333.951,Z 661.486,A -85,B 0,C 180,E1 -20374.36,E2 -20374.36} C_VEL
LIN {X 0,Y 335.16,Z 661.308,A -85,B 0,C 180,E1 -20374.67,E2 -20374.67} C_VEL
LIN {X 0,Y 337.514,Z 658.355,A -85,B 0,C 180,E1 -20375.055,E2 -20375.055} C_VEL
LIN {X 0,Y 341.352,Z 650.713,A -85,B 0,C 180,E1 -20375.463,E2 -20375.463} C_VEL
LIN {X 0,Y 345.98,Z 638.87,A -85,B 0,C 180,E1 -20375.768,E2 -20375.768} C_VEL
LIN {X 0,Y 349.083,Z 635.013,A -85,B 0,C 180,E1 -20376.263,E2 -20376.263} C_VEL
LIN {X 0,Y 353.01,Z 627.661,A -85,B 0,C 180,E1 -20376.702,E2 -20376.702} C_VEL
LIN {X 0,Y 357.945,Z 615.208,A -85,B 0,C 180,E1 -20377.062,E2 -20377.062} C_VEL
LIN {X 0,Y 359.438,Z 611.224,A -85,B 0,C 180,E1 -20377.157,E2 -20377.157} C_VEL
LIN {X 0,Y 363.279,Z 605.267,A -85,B 0,C 180,E1 -20377.665,E2 -20377.665} C_VEL
LIN {X 0,Y 367.78,Z 595.544,A -85,B 0,C 180,E1 -20378.096,E2 -20378.096} C_VEL
LIN {X 0,Y 373.457,Z 579.976,A -85,B 0,C 180,E1 -20378.474,E2 -20378.474} C_VEL
LIN {X 0,Y 377.822,Z 572.403,A -85,B 0,C 180,E1 -20378.991,E2 -20378.991} C_VEL
LIN {X 0,Y 382.721,Z 560.896,A -85,B 0,C 180,E1 -20379.422,E2 -20379.422} C_VEL
LIN {X 0,Y 384.053,Z 557.395,A -85,B 0,C 180,E1 -20379.524,E2 -20379.524} C_VEL
LIN {X 0,Y 377.738,Z 610.812,A -85,B 0,C 180,E1 -20380.896,E2 -20380.896} C_VEL
LIN {X 0,Y 371.828,Z 656.088,A -85,B 0,C 180,E1 -20382.302,E2 -20382.302} C_VEL
LIN {X 0,Y 367.183,Z 693.828,A -85,B 0,C 180,E1 -20383.787,E2 -20383.787} C_VEL
LIN {X 0,Y 363.852,Z 715.266,A -85,B 0,C 180,E1 -20384.908,E2 -20384.908} C_VEL
LIN {X 0,Y 359.715,Z 735.954,A -85,B 0,C 180,E1 -20386.28,E2 -20386.28} C_VEL
LIN {X 0,Y 354.966,Z 755.652,A -85,B 0,C 180,E1 -20387.901,E2 -20387.901} C_VEL
LIN {X 0,Y 349.776,Z 774.115,A -85,B 0,C 180,E1 -20389.755,E2 -20389.755} C_VEL
LIN {X 0,Y 344.215,Z 791.654,A -85,B 0,C 180,E1 -20391.882,E2 -20391.882} C_VEL
LIN {X 0,Y 338.433,Z 808.228,A -85,B 0,C 180,E1 -20394.302,E2 -20394.302} C_VEL
LIN {X 0,Y 332.607,Z 823.718,A -85,B 0,C 180,E1 -20397.035,E2 -20397.035} C_VEL
LIN {X 0,Y 327.217,Z 837.285,A -85,B 0,C 180,E1 -20399.924,E2 -20399.924} C_VEL
LIN {X 0,Y 321.954,Z 850.095,A -85,B 0,C 180,E1 -20403.235,E2 -20403.235} C_VEL
LIN {X 0,Y 317.521,Z 860.767,A -85,B 0,C 180,E1 -20406.623,E2 -20406.623} C_VEL
LIN {X 0,Y 313.74,Z 870.01,A -85,B 0,C 180,E1 -20410.256,E2 -20410.256} C_VEL
LIN {X 0,Y 310.66,Z 877.924,A -85,B 0,C 180,E1 -20414.231,E2 -20414.231} C_VEL
LIN {X 0,Y 308.519,Z 883.862,A -85,B 0,C 180,E1 -20418.218,E2 -20418.218} C_VEL
LIN {X 0,Y 307.222,Z 887.941,A -85,B 0,C 180,E1 -20422.143,E2 -20422.143} C_VEL
LIN {X 0,Y 306.564,Z 890.323,A -85,B 0,C 180,E1 -20425.885,E2 -20425.885} C_VEL
LIN {X 0,Y 306.339,Z 891.208,A -85,B 0,C 180,E1 -20429.813,E2 -20429.813} C_VEL
LIN {X 0,Y 306.489,Z 890.546,A -85,B 0,C 180,E1 -20433.554,E2 -20433.554} C_VEL
LIN {X 0,Y 307.114,Z 888.319,A -85,B 0,C 180,E1 -20437.483,E2 -20437.483} C_VEL
LIN {X 0,Y 308.332,Z 884.471,A -85,B 0,C 180,E1 -20441.409,E2 -20441.409} C_VEL
LIN {X 0,Y 310.224,Z 879.232,A -85,B 0,C 180,E1 -20445.134,E2 -20445.134} C_VEL
LIN {X 0,Y 313.037,Z 871.933,A -85,B 0,C 180,E1 -20449.014,E2 -20449.014} C_VEL
LIN {X 0,Y 316.625,Z 863.138,A -85,B 0,C 180,E1 -20452.661,E2 -20452.661} C_VEL
LIN {X 0,Y 321.17,Z 852.205,A -85,B 0,C 180,E1 -20456.282,E2 -20456.282} C_VEL
LIN {X 0,Y 326.231,Z 839.96,A -85,B 0,C 180,E1 -20459.568,E2 -20459.568} C_VEL
LIN {X 0,Y 331.829,Z 826.009,A -85,B 0,C 180,E1 -20462.641,E2 -20462.641} C_VEL
LIN {X 0,Y 336.78,Z 812.978,A -85,B 0,C 180,E1 -20465.029,E2 -20465.029} C_VEL
LIN {X 0,Y 337.941,Z 807.852,A -85,B 0,C 180,E1 -20466,E2 -20466} C_VEL
LIN {X 0,Y 338.029,Z 795.096,A -85,B 0,C 180,E1 -20468.628,E2 -20468.628} C_VEL
LIN {X 0,Y 339.242,Z 789.378,A -85,B 0,C 180,E1 -20469.505,E2 -20469.505} C_VEL
LIN {X 0,Y 344.718,Z 772.32,A -85,B 0,C 180,E1 -20471.524,E2 -20471.524} C_VEL
LIN {X 0,Y 349.871,Z 754.202,A -85,B 0,C 180,E1 -20473.306,E2 -20473.306} C_VEL
LIN {X 0,Y 354.503,Z 735.274,A -85,B 0,C 180,E1 -20474.84,E2 -20474.84} C_VEL
LIN {X 0,Y 358.506,Z 715.628,A -85,B 0,C 180,E1 -20476.135,E2 -20476.135} C_VEL
LIN {X 0,Y 361.748,Z 695.38,A -85,B 0,C 180,E1 -20477.199,E2 -20477.199} C_VEL
LIN {X 0,Y 366.788,Z 656.184,A -85,B 0,C 180,E1 -20478.757,E2 -20478.757} C_VEL
LIN {X 0,Y 372.959,Z 610.416,A -85,B 0,C 180,E1 -20480.183,E2 -20480.183} C_VEL
LIN {X 0,Y 379.409,Z 556.738,A -85,B 0,C 180,E1 -20481.555,E2 -20481.555} C_VEL
LIN {X 0,Y 384.354,Z 505.086,A -85,B 0,C 180,E1 -20482.666,E2 -20482.666} C_VEL
LIN {X 0,Y 389.545,Z 434.203,A -85,B 0,C 180,E1 -20483.954,E2 -20483.954} C_VEL
LIN {X 0,Y 396.422,Z 403.987,A -85,B 0,C 180,E1 -20484.983,E2 -20484.983} C_VEL
LIN {X 0,Y 391.293,Z 388.296,A -85,B 0,C 180,E1 -20487.76,E2 -20487.76} C_VEL
LIN {X 0,Y 386.296,Z 374.674,A -85,B 0,C 180,E1 -20490.541,E2 -20490.541} C_VEL
LIN {X 0,Y 380.965,Z 361.708,A -85,B 0,C 180,E1 -20493.627,E2 -20493.627} C_VEL
LIN {X 0,Y 375.965,Z 350.58,A -85,B 0,C 180,E1 -20496.738,E2 -20496.738} C_VEL
LIN {X 0,Y 371.595,Z 341.709,A -85,B 0,C 180,E1 -20499.689,E2 -20499.689} C_VEL
LIN {X 0,Y 367.995,Z 334.569,A -85,B 0,C 180,E1 -20502.446,E2 -20502.446} C_VEL
LIN {X 0,Y 365.073,Z 329.366,A -85,B 0,C 180,E1 -20504.837,E2 -20504.837} C_VEL
LIN {X 0,Y 362.77,Z 325.055,A -85,B 0,C 180,E1 -20507.099,E2 -20507.099} C_VEL
LIN {X 0,Y 360.543,Z 320.629,A -85,B 0,C 180,E1 -20509.857,E2 -20509.857} C_VEL
LIN {X 0,Y 358.077,Z 316.846,A -85,B 0,C 180,E1 -20513.426,E2 -20513.426} C_VEL
LIN {X 0,Y 357.526,Z 314.915,A -85,B 0,C 180,E1 -20514.865,E2 -20514.865} C_VEL
LIN {X 0,Y 356.253,Z 313.222,A -85,B 0,C 180,E1 -20521.126,E2 -20521.126} C_VEL
LIN {X 0,Y 357.213,Z 313.883,A -85,B 0,C 180,E1 -20525.461,E2 -20525.461} C_VEL
LIN {X 0,Y 359.144,Z 315.45,A -85,B 0,C 180,E1 -20528.727,E2 -20528.727} C_VEL
LIN {X 0,Y 361.232,Z 328.608,A -85,B 0,C 180,E1 -20533.323,E2 -20533.323} C_VEL
LIN {X 0,Y 364.98,Z 342.359,A -85,B 0,C 180,E1 -20537.374,E2 -20537.374} C_VEL
LIN {X 0,Y 371.783,Z 362.34,A -85,B 0,C 180,E1 -20542.327,E2 -20542.327} C_VEL
LIN {X 0,Y 375.954,Z 373.486,A -85,B 0,C 180,E1 -20544.681,E2 -20544.681} C_VEL
LIN {X 0,Y 383.974,Z 396.356,A -85,B 0,C 180,E1 -20548.609,E2 -20548.609} C_VEL
LIN {X 0,Y 385.536,Z 399.783,A -85,B 0,C 180,E1 -20549.139,E2 -20549.139} C_VEL
LIN {X 0,Y 385.698,Z 401.009,A -85,B 0,C 180,E1 -20549.205,E2 -20549.205} C_VEL
LIN {X 0,Y 357.72,Z 692.574,A -85,B 0,C 180,E1 -20556.448,E2 -20556.448} C_VEL
LIN {X 0,Y 354.365,Z 717.163,A -85,B 0,C 180,E1 -20557.334,E2 -20557.334} C_VEL
LIN {X 0,Y 350.151,Z 742.267,A -85,B 0,C 180,E1 -20558.516,E2 -20558.516} C_VEL
LIN {X 0,Y 341.188,Z 789.824,A -85,B 0,C 180,E1 -20561.389,E2 -20561.389} C_VEL
LIN {X 0,Y 336.274,Z 814.779,A -85,B 0,C 180,E1 -20563.24,E2 -20563.24} C_VEL
LIN {X 0,Y 331.992,Z 833.623,A -85,B 0,C 180,E1 -20564.946,E2 -20564.946} C_VEL
LIN {X 0,Y 327.337,Z 851.652,A -85,B 0,C 180,E1 -20566.944,E2 -20566.944} C_VEL
LIN {X 0,Y 322.418,Z 868.707,A -85,B 0,C 180,E1 -20569.246,E2 -20569.246} C_VEL
LIN {X 0,Y 317.387,Z 884.838,A -85,B 0,C 180,E1 -20571.868,E2 -20571.868} C_VEL
LIN {X 0,Y 312.552,Z 900.015,A -85,B 0,C 180,E1 -20574.842,E2 -20574.842} C_VEL
LIN {X 0,Y 308.132,Z 913.728,A -85,B 0,C 180,E1 -20578.067,E2 -20578.067} C_VEL
LIN {X 0,Y 304.347,Z 925.934,A -85,B 0,C 180,E1 -20581.551,E2 -20581.551} C_VEL
LIN {X 0,Y 301.157,Z 937.218,A -85,B 0,C 180,E1 -20585.48,E2 -20585.48} C_VEL
LIN {X 0,Y 299.026,Z 946.472,A -85,B 0,C 180,E1 -20589.445,E2 -20589.445} C_VEL
LIN {X 0,Y 297.838,Z 953.879,A -85,B 0,C 180,E1 -20593.42,E2 -20593.42} C_VEL
LIN {X 0,Y 297.438,Z 959.796,A -85,B 0,C 180,E1 -20597.576,E2 -20597.576} C_VEL
LIN {X 0,Y 297.642,Z 965.012,A -85,B 0,C 180,E1 -20602.472,E2 -20602.472} C_VEL
LIN {X 0,Y 297.86,Z 968.051,A -85,B 0,C 180,E1 -20605.958,E2 -20605.958} C_VEL
LIN {X 0,Y 297.91,Z 969.914,A -85,B 0,C 180,E1 -20609.616,E2 -20609.616} C_VEL
LIN {X 0,Y 297.666,Z 970.309,A -85,B 0,C 180,E1 -20613.274,E2 -20613.274} C_VEL
LIN {X 0,Y 297.231,Z 969.515,A -85,B 0,C 180,E1 -20616.762,E2 -20616.762} C_VEL
LIN {X 0,Y 296.919,Z 967.523,A -85,B 0,C 180,E1 -20620.478,E2 -20620.478} C_VEL
LIN {X 0,Y 297.166,Z 963.42,A -85,B 0,C 180,E1 -20625.216,E2 -20625.216} C_VEL
LIN {X 0,Y 298.467,Z 957.805,A -85,B 0,C 180,E1 -20629.777,E2 -20629.777} C_VEL
LIN {X 0,Y 301.528,Z 949.695,A -85,B 0,C 180,E1 -20634.907,E2 -20634.907} C_VEL
LIN {X 0,Y 306.392,Z 940.012,A -85,B 0,C 180,E1 -20639.764,E2 -20639.764} C_VEL
LIN {X 0,Y 313.805,Z 927.706,A -85,B 0,C 180,E1 -20644.775,E2 -20644.775} C_VEL
LIN {X 0,Y 323.243,Z 913.972,A -85,B 0,C 180,E1 -20649.356,E2 -20649.356} C_VEL
LIN {X 0,Y 334.892,Z 898.353,A -85,B 0,C 180,E1 -20653.606,E2 -20653.606} C_VEL
LIN {X 0,Y 348.712,Z 880.922,A -85,B 0,C 180,E1 -20657.47,E2 -20657.47} C_VEL
LIN {X 0,Y 364.003,Z 862.509,A -85,B 0,C 180,E1 -20660.772,E2 -20660.772} C_VEL
LIN {X 0,Y 374.502,Z 850.087,A -85,B 0,C 180,E1 -20662.646,E2 -20662.646} C_VEL
LIN {X 0,Y 359.179,Z 863.893,A -85,B 0,C 180,E1 -20665.396,E2 -20665.396} C_VEL
LIN {X 0,Y 345.39,Z 876.409,A -85,B 0,C 180,E1 -20668.594,E2 -20668.594} C_VEL
LIN {X 0,Y 334.044,Z 886.682,A -85,B 0,C 180,E1 -20671.969,E2 -20671.969} C_VEL
LIN {X 0,Y 324.816,Z 894.747,A -85,B 0,C 180,E1 -20675.444,E2 -20675.444} C_VEL
LIN {X 0,Y 317.429,Z 900.711,A -85,B 0,C 180,E1 -20678.955,E2 -20678.955} C_VEL
LIN {X 0,Y 311.375,Z 904.852,A -85,B 0,C 180,E1 -20682.624,E2 -20682.624} C_VEL
LIN {X 0,Y 306.614,Z 907.076,A -85,B 0,C 180,E1 -20686.42,E2 -20686.42} C_VEL
LIN {X 0,Y 303.223,Z 907.337,A -85,B 0,C 180,E1 -20690.127,E2 -20690.127} C_VEL
LIN {X 0,Y 300.934,Z 905.842,A -85,B 0,C 180,E1 -20693.705,E2 -20693.705} C_VEL
LIN {X 0,Y 299.448,Z 902.582,A -85,B 0,C 180,E1 -20697.321,E2 -20697.321} C_VEL
LIN {X 0,Y 298.646,Z 897.473,A -85,B 0,C 180,E1 -20700.959,E2 -20700.959} C_VEL
LIN {X 0,Y 298.396,Z 890.829,A -85,B 0,C 180,E1 -20704.42,E2 -20704.42} C_VEL
LIN {X 0,Y 298.637,Z 882.294,A -85,B 0,C 180,E1 -20707.89,E2 -20707.89} C_VEL
LIN {X 0,Y 299.334,Z 872.343,A -85,B 0,C 180,E1 -20711.171,E2 -20711.171} C_VEL
LIN {X 0,Y 300.57,Z 860.253,A -85,B 0,C 180,E1 -20714.448,E2 -20714.448} C_VEL
LIN {X 0,Y 302.28,Z 846.733,A -85,B 0,C 180,E1 -20717.519,E2 -20717.519} C_VEL
LIN {X 0,Y 304.571,Z 830.787,A -85,B 0,C 180,E1 -20720.565,E2 -20720.565} C_VEL
LIN {X 0,Y 307.18,Z 813.682,A -85,B 0,C 180,E1 -20723.297,E2 -20723.297} C_VEL
